LIN {X 0.010,Y -561.070,Z 1059.302,A 0.000,B 0.000,C 90.000,E1 90.286} C_DIS
LIN {X -0.066,Y -561.534,Z 1059.294,A 0.000,B 0.000,C 90.000,E1 88.912} C_DIS
LIN {X -0.024,Y -562.090,Z 1059.285,A 0.000,B 0.000,C 90.000,E1 87.249} C_DIS
LIN {X 0.060,Y -562.761,Z 1059.276,A 0.000,B 0.000,C 90.000,E1 85.584} C_DIS
LIN {X 0.063,Y -563.206,Z 1059.268,A 0.000,B 0.000,C 90.000,E1 84.204} C_DIS
LIN {X -0.191,Y -563.676,Z 1059.257,A 0.000,B 0.000,C 90.000,E1 82.299} C_DIS
LIN {X 0.040,Y -564.205,Z 1059.248,A 0.000,B 0.000,C 90.000,E1 80.622} C_DIS
LIN {X 0.142,Y -565.085,Z 1059.236,A 0.000,B 0.000,C 90.000,E1 78.409} C_DIS
LIN {X -0.127,Y -565.808,Z 1059.228,A 0.000,B 0.000,C 90.000,E1 77.061} C_DIS
LIN {X 0.019,Y -567.276,Z 1059.214,A 0.000,B 0.000,C 90.000,E1 74.574} C_DIS
LIN {X -0.132,Y -568.746,Z 1059.204,A 0.000,B 0.000,C 90.000,E1 72.670} C_DIS
LIN {X -0.096,Y -570.540,Z 1059.192,A 0.000,B 0.000,C 90.000,E1 70.477} C_DIS
LIN {X -0.152,Y -571.474,Z 1059.185,A 0.000,B 0.000,C 90.000,E1 69.390} C_DIS
LIN {X -0.198,Y -572.979,Z 1059.175,A 0.000,B 0.000,C 90.000,E1 67.486} C_DIS
LIN {X -0.127,Y -574.101,Z 1059.166,A 0.000,B 0.000,C 90.000,E1 65.845} C_DIS
LIN {X -0.178,Y -575.248,Z 1059.155,A 0.000,B 0.000,C 90.000,E1 63.948} C_DIS
LIN {X 0.199,Y -576.123,Z 1059.146,A 0.000,B 0.000,C 90.000,E1 62.281} C_DIS
LIN {X 0.224,Y -576.847,Z 1059.139,A 0.000,B 0.000,C 90.000,E1 60.923} C_DIS
LIN {X -0.113,Y -577.556,Z 1059.130,A 0.000,B 0.000,C 90.000,E1 59.331} C_DIS
LIN {X -0.133,Y -578.213,Z 1059.121,A 0.000,B 0.000,C 90.000,E1 57.709} C_DIS
LIN {X -0.146,Y -578.878,Z 1059.112,A 0.000,B 0.000,C 90.000,E1 56.087} C_DIS
LIN {X -0.145,Y -579.399,Z 1059.101,A 0.000,B 0.000,C 90.000,E1 54.196} C_DIS
LIN {X 0.187,Y -579.510,Z 1059.098,A 0.000,B 0.000,C 90.000,E1 53.623} C_DIS
LIN {X 0.206,Y -579.521,Z 1059.091,A 0.000,B 0.000,C 90.000,E1 52.271} C_DIS
LIN {X 0.246,Y -579.470,Z 1059.086,A 0.000,B 0.000,C 90.000,E1 51.457} C_DIS
LIN {X -0.077,Y -579.230,Z 1059.082,A 0.000,B 0.000,C 90.000,E1 50.678} C_DIS
LIN {X 0.207,Y -578.665,Z 1059.074,A 0.000,B 0.000,C 90.000,E1 49.299} C_DIS
LIN {X 0.105,Y -578.034,Z 1059.067,A 0.000,B 0.000,C 90.000,E1 47.957} C_DIS
LIN {X -0.198,Y -577.318,Z 1059.061,A 0.000,B 0.000,C 90.000,E1 46.905} C_DIS
LIN {X 0.198,Y -576.692,Z 1059.056,A 0.000,B 0.000,C 90.000,E1 46.053} C_DIS
LIN {X 0.169,Y -575.894,Z 1059.052,A 0.000,B 0.000,C 90.000,E1 45.243} C_DIS
LIN {X 0.374,Y -574.257,Z 1059.044,A 0.000,B 0.000,C 90.000,E1 43.866} C_DIS
LIN {X 0.147,Y -572.209,Z 1059.036,A 0.000,B 0.000,C 90.000,E1 42.528} C_DIS
LIN {X -0.321,Y -570.874,Z 1059.032,A 0.000,B 0.000,C 90.000,E1 41.757} C_DIS
LIN {X 0.000,Y -569.379,Z 1059.027,A 0.000,B 0.000,C 90.000,E1 40.906} C_DIS
LIN {X -0.265,Y -566.286,Z 1059.020,A 0.000,B 0.000,C 90.000,E1 39.564} C_DIS
LIN {X -0.145,Y -562.491,Z 1059.012,A 0.000,B 0.000,C 90.000,E1 38.177} C_DIS
LIN {X 0.162,Y -559.808,Z 1059.007,A 0.000,B 0.000,C 90.000,E1 37.317} C_DIS
LIN {X -0.096,Y -557.923,Z 1059.004,A 0.000,B 0.000,C 90.000,E1 36.790} C_DIS
LIN {X 0.076,Y -555.871,Z 1059.001,A 0.000,B 0.000,C 90.000,E1 36.217} C_DIS
LIN {X -0.017,Y -552.360,Z 1058.997,A 0.000,B 0.000,C 90.000,E1 35.391} C_DIS
LIN {X -0.014,Y -549.197,Z 1058.993,A 0.000,B 0.000,C 90.000,E1 34.692} C_DIS
LIN {X -0.004,Y -544.551,Z 1058.987,A 0.000,B 0.000,C 90.000,E1 33.706} C_DIS
LIN {X 0.251,Y -538.674,Z 1058.981,A 0.000,B 0.000,C 90.000,E1 32.546} C_DIS
LIN {X -0.167,Y -534.651,Z 1058.977,A 0.000,B 0.000,C 90.000,E1 31.878} C_DIS
LIN {X -0.034,Y -529.513,Z 1058.972,A 0.000,B 0.000,C 90.000,E1 31.003} C_DIS
LIN {X 0.196,Y -524.774,Z 1058.968,A 0.000,B 0.000,C 90.000,E1 30.256} C_DIS
LIN {X -0.212,Y -517.541,Z 1058.963,A 0.000,B 0.000,C 90.000,E1 29.283} C_DIS
LIN {X -0.104,Y -511.824,Z 1058.958,A 0.000,B 0.000,C 90.000,E1 28.537} C_DIS
LIN {X 0.091,Y -506.976,Z 1058.955,A 0.000,B 0.000,C 90.000,E1 27.924} C_DIS
LIN {X -0.206,Y -503.132,Z 1058.953,A 0.000,B 0.000,C 90.000,E1 27.513} C_DIS
LIN {X 0.157,Y -496.395,Z 1058.949,A 0.000,B 0.000,C 90.000,E1 26.744} C_DIS
LIN {X 0.074,Y -490.864,Z 1058.946,A 0.000,B 0.000,C 90.000,E1 26.181} C_DIS
LIN {X 0.160,Y -482.412,Z 1058.941,A 0.000,B 0.000,C 90.000,E1 25.335} C_DIS
LIN {X 0.165,Y -473.830,Z 1058.936,A 0.000,B 0.000,C 90.000,E1 24.515} C_DIS
LIN {X 0.287,Y -466.468,Z 1058.933,A 0.000,B 0.000,C 90.000,E1 23.823} C_DIS
LIN {X 0.179,Y -456.040,Z 1058.928,A 0.000,B 0.000,C 90.000,E1 22.950} C_DIS
LIN {X -0.144,Y -446.987,Z 1058.923,A 0.000,B 0.000,C 90.000,E1 22.206} C_DIS
LIN {X 0.000,Y -427.675,Z 1058.914,A 0.000,B 0.000,C 90.000,E1 20.429} C_DIS
LIN {X -0.121,Y -416.146,Z 1058.907,A 0.000,B 0.000,C 90.000,E1 19.268} C_DIS
LIN {X -0.045,Y -403.587,Z 1058.899,A 0.000,B 0.000,C 90.000,E1 17.819} C_DIS
LIN {X -0.132,Y -398.339,Z 1058.895,A 0.000,B 0.000,C 90.000,E1 17.149} C_DIS
LIN {X -0.196,Y -395.334,Z 1058.893,A 0.000,B 0.000,C 90.000,E1 16.677} C_DIS
LIN {X -0.074,Y -394.456,Z 1058.892,A 0.000,B 0.000,C 90.000,E1 16.496} C_DIS
LIN {X -0.121,Y -392.733,Z 1058.889,A 0.000,B 0.000,C 90.000,E1 16.079} C_DIS
LIN {X 0.029,Y -391.733,Z 1058.886,A 0.000,B 0.000,C 90.000,E1 15.481} C_DIS
LIN {X -0.132,Y -391.606,Z 1058.883,A 0.000,B 0.000,C 90.000,E1 14.883} C_DIS
LIN {X 0.221,Y -392.903,Z 1058.875,A 0.000,B 0.000,C 90.000,E1 13.411} C_DIS
LIN {X -0.007,Y -398.590,Z 1058.853,A 0.000,B 0.000,C 90.000,E1 9.557} C_DIS
LIN {X -0.170,Y -403.813,Z 1058.838,A 0.000,B 0.000,C 90.000,E1 6.777} C_DIS
LIN {X 0.136,Y -409.152,Z 1058.824,A 0.000,B 0.000,C 90.000,E1 4.302} C_DIS
LIN {X 0.131,Y -411.130,Z 1058.820,A 0.000,B 0.000,C 90.000,E1 3.612} C_DIS
LIN {X -0.082,Y -411.998,Z 1058.819,A 0.000,B 0.000,C 90.000,E1 3.383} C_DIS
LIN {X -0.064,Y -415.403,Z 1058.816,A 0.000,B 0.000,C 90.000,E1 2.808} C_DIS
LIN {X -0.061,Y -416.570,Z 1058.815,A 0.000,B 0.000,C 90.000,E1 2.636} C_DIS
LIN {X -0.059,Y -418.064,Z 1058.814,A 0.000,B 0.000,C 90.000,E1 2.465} C_DIS
LIN {X 0.191,Y -421.574,Z 1058.812,A 0.000,B 0.000,C 90.000,E1 2.121} C_DIS
LIN {X 0.026,Y -423.409,Z 1058.811,A 0.000,B 0.000,C 90.000,E1 2.007} C_DIS
LIN {X 0.078,Y -434.006,Z 1058.807,A 0.000,B 0.000,C 90.000,E1 1.318} C_DIS
LIN {X 0.086,Y -456.510,Z 1058.799,A 0.000,B 0.000,C 90.000,E1 359.885} C_DIS
LIN {X 0.073,Y -471.379,Z 1058.794,A 0.000,B 0.000,C 90.000,E1 358.969} C_DIS
LIN {X 0.112,Y -484.516,Z 1058.790,A 0.000,B 0.000,C 90.000,E1 358.165} C_DIS
LIN {X -0.130,Y -495.813,Z 1058.786,A 0.000,B 0.000,C 90.000,E1 357.478} C_DIS
LIN {X -0.216,Y -503.707,Z 1058.783,A 0.000,B 0.000,C 90.000,E1 356.963} C_DIS
LIN {X 0.045,Y -511.351,Z 1058.780,A 0.000,B 0.000,C 90.000,E1 356.388} C_DIS
LIN {X 0.098,Y -518.758,Z 1058.777,A 0.000,B 0.000,C 90.000,E1 355.812} C_DIS
LIN {X -0.107,Y -524.566,Z 1058.774,A 0.000,B 0.000,C 90.000,E1 355.355} C_DIS
LIN {X 0.229,Y -530.049,Z 1058.771,A 0.000,B 0.000,C 90.000,E1 354.837} C_DIS
LIN {X 0.199,Y -535.561,Z 1058.769,A 0.000,B 0.000,C 90.000,E1 354.318} C_DIS
LIN {X -0.151,Y -541.884,Z 1058.765,A 0.000,B 0.000,C 90.000,E1 353.685} C_DIS
LIN {X 0.069,Y -546.768,Z 1058.762,A 0.000,B 0.000,C 90.000,E1 353.109} C_DIS
LIN {X 0.008,Y -552.220,Z 1058.758,A 0.000,B 0.000,C 90.000,E1 352.413} C_DIS
LIN {X 0.161,Y -556.239,Z 1058.755,A 0.000,B 0.000,C 90.000,E1 351.837} C_DIS
LIN {X 0.178,Y -560.694,Z 1058.751,A 0.000,B 0.000,C 90.000,E1 351.141} C_DIS
LIN {X -0.168,Y -564.024,Z 1058.748,A 0.000,B 0.000,C 90.000,E1 350.622} C_DIS
LIN {X -0.088,Y -567.760,Z 1058.744,A 0.000,B 0.000,C 90.000,E1 349.926} C_DIS
LIN {X 0.134,Y -571.203,Z 1058.740,A 0.000,B 0.000,C 90.000,E1 349.218} C_DIS
LIN {X 0.044,Y -575.033,Z 1058.736,A 0.000,B 0.000,C 90.000,E1 348.409} C_DIS
LIN {X 0.204,Y -580.307,Z 1058.729,A 0.000,B 0.000,C 90.000,E1 347.173} C_DIS
LIN {X -0.019,Y -584.594,Z 1058.723,A 0.000,B 0.000,C 90.000,E1 346.117} C_DIS
LIN {X 0.204,Y -589.665,Z 1058.715,A 0.000,B 0.000,C 90.000,E1 344.755} C_DIS
LIN {X -0.056,Y -594.516,Z 1058.708,A 0.000,B 0.000,C 90.000,E1 343.449} C_DIS
LIN {X 0.229,Y -598.177,Z 1058.702,A 0.000,B 0.000,C 90.000,E1 342.362} C_DIS
LIN {X 0.003,Y -601.590,Z 1058.696,A 0.000,B 0.000,C 90.000,E1 341.329} C_DIS
LIN {X -0.091,Y -603.905,Z 1058.692,A 0.000,B 0.000,C 90.000,E1 340.550} C_DIS
LIN {X 0.038,Y -606.170,Z 1058.688,A 0.000,B 0.000,C 90.000,E1 339.752} C_DIS
LIN {X -0.141,Y -609.589,Z 1058.680,A 0.000,B 0.000,C 90.000,E1 338.465} C_DIS
LIN {X 0.049,Y -611.504,Z 1058.676,A 0.000,B 0.000,C 90.000,E1 337.667} C_DIS
LIN {X 0.187,Y -614.433,Z 1058.669,A 0.000,B 0.000,C 90.000,E1 336.357} C_DIS
LIN {X -0.191,Y -616.880,Z 1058.662,A 0.000,B 0.000,C 90.000,E1 335.101} C_DIS
LIN {X 0.291,Y -618.961,Z 1058.654,A 0.000,B 0.000,C 90.000,E1 333.768} C_DIS
LIN {X 0.251,Y -620.720,Z 1058.647,A 0.000,B 0.000,C 90.000,E1 332.487} C_DIS
LIN {X -0.316,Y -622.272,Z 1058.640,A 0.000,B 0.000,C 90.000,E1 331.257} C_DIS
LIN {X -0.017,Y -623.078,Z 1058.636,A 0.000,B 0.000,C 90.000,E1 330.461} C_DIS
LIN {X -0.243,Y -623.905,Z 1058.630,A 0.000,B 0.000,C 90.000,E1 329.459} C_DIS
LIN {X 0.075,Y -624.459,Z 1058.625,A 0.000,B 0.000,C 90.000,E1 328.408} C_DIS
LIN {X -0.134,Y -624.866,Z 1058.620,A 0.000,B 0.000,C 90.000,E1 327.661} C_DIS
LIN {X -0.006,Y -624.992,Z 1058.615,A 0.000,B 0.000,C 90.000,E1 326.628} C_DIS
LIN {X 0.126,Y -624.944,Z 1058.609,A 0.000,B 0.000,C 90.000,E1 325.595} C_DIS
LIN {X 0.084,Y -624.711,Z 1058.602,A 0.000,B 0.000,C 90.000,E1 324.322} C_DIS
LIN {X 0.178,Y -624.070,Z 1058.591,A 0.000,B 0.000,C 90.000,E1 322.271} C_DIS
LIN {X -0.171,Y -623.409,Z 1058.576,A 0.000,B 0.000,C 90.000,E1 319.747} C_DIS
LIN {X 0.056,Y -623.246,Z 1058.569,A 0.000,B 0.000,C 90.000,E1 318.447} C_DIS
LIN {X 0.098,Y -623.046,Z 1058.565,A 0.000,B 0.000,C 90.000,E1 317.676} C_DIS
LIN {X -0.110,Y -622.573,Z 1058.554,A 0.000,B 0.000,C 90.000,E1 315.648} C_DIS
LIN {X -0.212,Y -622.237,Z 1058.544,A 0.000,B 0.000,C 90.000,E1 313.866} C_DIS
LIN {X -0.185,Y -622.125,Z 1058.539,A 0.000,B 0.000,C 90.000,E1 313.095} C_DIS
LIN {X 0.433,Y -621.704,Z 1058.532,A 0.000,B 0.000,C 90.000,E1 311.757} C_DIS
LIN {X -0.254,Y -621.130,Z 1058.525,A 0.000,B 0.000,C 90.000,E1 310.539} C_DIS
LIN {X 0.066,Y -621.133,Z 1058.524,A 0.000,B 0.000,C 90.000,E1 310.253} C_DIS
LIN {X 0.235,Y -620.888,Z 1058.521,A 0.000,B 0.000,C 90.000,E1 309.725} C_DIS
LIN {X 0.078,Y -620.896,Z 1058.519,A 0.000,B 0.000,C 90.000,E1 309.483} C_DIS
LIN {X -0.284,Y -620.114,Z 1058.505,A 0.000,B 0.000,C 90.000,E1 306.950} C_DIS
LIN {X -0.138,Y -620.085,Z 1058.502,A 0.000,B 0.000,C 90.000,E1 306.423} C_DIS
LIN {X -0.083,Y -619.896,Z 1058.497,A 0.000,B 0.000,C 90.000,E1 305.391} C_DIS
LIN {X 0.238,Y -619.761,Z 1058.495,A 0.000,B 0.000,C 90.000,E1 305.105} C_DIS
LIN {X 0.013,Y -619.990,Z 1058.492,A 0.000,B 0.000,C 90.000,E1 304.612} C_DIS
LIN {X 0.393,Y -619.920,Z 1058.485,A 0.000,B 0.000,C 90.000,E1 303.293} C_DIS
LIN {X -0.151,Y -619.823,Z 1058.484,A 0.000,B 0.000,C 90.000,E1 303.086} C_DIS
LIN {X 0.139,Y -620.073,Z 1058.481,A 0.000,B 0.000,C 90.000,E1 302.546} C_DIS
LIN {X -0.113,Y -620.174,Z 1058.477,A 0.000,B 0.000,C 90.000,E1 301.799} C_DIS
LIN {X 0.165,Y -620.036,Z 1058.472,A 0.000,B 0.000,C 90.000,E1 301.003} C_DIS
LIN {X -0.090,Y -620.335,Z 1058.468,A 0.000,B 0.000,C 90.000,E1 300.256} C_DIS
LIN {X 0.167,Y -620.678,Z 1058.460,A 0.000,B 0.000,C 90.000,E1 298.693} C_DIS
LIN {X -0.120,Y -620.453,Z 1058.451,A 0.000,B 0.000,C 90.000,E1 297.180} C_DIS
LIN {X -0.149,Y -619.802,Z 1058.444,A 0.000,B 0.000,C 90.000,E1 295.899} C_DIS
LIN {X 0.115,Y -618.831,Z 1058.438,A 0.000,B 0.000,C 90.000,E1 294.847} C_DIS
LIN {X 0.082,Y -617.754,Z 1058.434,A 0.000,B 0.000,C 90.000,E1 294.079} C_DIS
LIN {X -0.236,Y -615.850,Z 1058.428,A 0.000,B 0.000,C 90.000,E1 293.078} C_DIS
LIN {X 0.281,Y -614.623,Z 1058.425,A 0.000,B 0.000,C 90.000,E1 292.514} C_DIS
LIN {X -0.014,Y -612.935,Z 1058.422,A 0.000,B 0.000,C 90.000,E1 292.025} C_DIS
LIN {X -0.050,Y -611.999,Z 1058.421,A 0.000,B 0.000,C 90.000,E1 291.770} C_DIS
LIN {X 0.210,Y -609.689,Z 1058.418,A 0.000,B 0.000,C 90.000,E1 291.227} C_DIS
LIN {X -0.112,Y -606.397,Z 1058.415,A 0.000,B 0.000,C 90.000,E1 290.737} C_DIS
LIN {X -0.287,Y -601.104,Z 1058.412,A 0.000,B 0.000,C 90.000,E1 290.248} C_DIS
LIN {X -0.092,Y -596.948,Z 1058.410,A 0.000,B 0.000,C 90.000,E1 289.866} C_DIS
LIN {X -0.208,Y -595.289,Z 1058.410,A 0.000,B 0.000,C 90.000,E1 289.758} C_DIS
LIN {X 0.152,Y -588.650,Z 1058.407,A 0.000,B 0.000,C 90.000,E1 289.322} C_DIS
LIN {X 0.358,Y -581.461,Z 1058.406,A 0.000,B 0.000,C 90.000,E1 288.960} C_DIS
LIN {X 0.216,Y -570.740,Z 1058.403,A 0.000,B 0.000,C 90.000,E1 288.544} C_DIS
LIN {X -0.092,Y -560.846,Z 1058.402,A 0.000,B 0.000,C 90.000,E1 288.362} C_DIS
LIN {X -0.097,Y -556.775,Z 1058.402,A 0.000,B 0.000,C 90.000,E1 288.290} C_DIS
LIN {X 0.284,Y -550.568,Z 1058.401,A 0.000,B 0.000,C 90.000,E1 288.236} C_DIS
LIN {X -0.233,Y -547.940,Z 1058.401,A 0.000,B 0.000,C 90.000,E1 288.236} C_DIS
LIN {X 0.243,Y -547.765,Z 1058.401,A 0.000,B 0.000,C 90.000,E1 288.181} C_DIS
LIN {X -0.099,Y -546.592,Z 1058.400,A 0.000,B 0.000,C 90.000,E1 287.946} C_DIS
LIN {X 0.275,Y -546.226,Z 1058.399,A 0.000,B 0.000,C 90.000,E1 287.819} C_DIS
LIN {X -0.166,Y -545.992,Z 1058.398,A 0.000,B 0.000,C 90.000,E1 287.583} C_DIS
LIN {X 0.079,Y -545.427,Z 1058.396,A 0.000,B 0.000,C 90.000,E1 287.275} C_DIS
LIN {X 0.231,Y -544.728,Z 1058.382,A 0.000,B 0.000,C 90.000,E1 284.717} C_DIS
LIN {X -0.256,Y -544.250,Z 1058.374,A 0.000,B 0.000,C 90.000,E1 283.355} C_DIS
LIN {X 0.186,Y -543.503,Z 1058.366,A 0.000,B 0.000,C 90.000,E1 281.895} C_DIS
LIN {X 0.170,Y -542.509,Z 1058.357,A 0.000,B 0.000,C 90.000,E1 280.197} C_DIS
LIN {X 0.027,Y -541.501,Z 1058.347,A 0.000,B 0.000,C 90.000,E1 278.511} C_DIS
LIN {X -0.221,Y -540.467,Z 1058.338,A 0.000,B 0.000,C 90.000,E1 276.834} C_DIS
LIN {X -0.084,Y -539.816,Z 1058.332,A 0.000,B 0.000,C 90.000,E1 275.682} C_DIS
LIN {X 0.109,Y -538.669,Z 1058.321,A 0.000,B 0.000,C 90.000,E1 273.669} C_DIS
LIN {X 0.230,Y -537.557,Z 1058.309,A 0.000,B 0.000,C 90.000,E1 271.661} C_DIS
LIN {X 0.266,Y -536.897,Z 1058.303,A 0.000,B 0.000,C 90.000,E1 270.516} C_DIS
LIN {X -0.228,Y -535.841,Z 1058.294,A 0.000,B 0.000,C 90.000,E1 268.854} C_DIS
LIN {X -0.200,Y -535.169,Z 1058.287,A 0.000,B 0.000,C 90.000,E1 267.707} C_DIS
LIN {X -0.183,Y -534.244,Z 1058.279,A 0.000,B 0.000,C 90.000,E1 266.274} C_DIS
LIN {X -0.152,Y -533.229,Z 1058.271,A 0.000,B 0.000,C 90.000,E1 264.837} C_DIS
LIN {X -0.084,Y -532.096,Z 1058.263,A 0.000,B 0.000,C 90.000,E1 263.394} C_DIS
LIN {X -0.038,Y -531.301,Z 1058.259,A 0.000,B 0.000,C 90.000,E1 262.527} C_DIS
LIN {X 0.031,Y -528.529,Z 1058.244,A 0.000,B 0.000,C 90.000,E1 259.926} C_DIS
LIN {X 0.172,Y -526.943,Z 1058.236,A 0.000,B 0.000,C 90.000,E1 258.465} C_DIS
LIN {X -0.232,Y -525.359,Z 1058.228,A 0.000,B 0.000,C 90.000,E1 257.061} C_DIS
LIN {X 0.112,Y -523.228,Z 1058.217,A 0.000,B 0.000,C 90.000,E1 254.991} C_DIS
LIN {X -0.099,Y -521.731,Z 1058.209,A 0.000,B 0.000,C 90.000,E1 253.559} C_DIS
LIN {X 0.173,Y -520.525,Z 1058.202,A 0.000,B 0.000,C 90.000,E1 252.362} C_DIS
LIN {X 0.210,Y -518.553,Z 1058.192,A 0.000,B 0.000,C 90.000,E1 250.604} C_DIS
LIN {X -0.151,Y -516.089,Z 1058.181,A 0.000,B 0.000,C 90.000,E1 248.592} C_DIS
LIN {X 0.027,Y -514.095,Z 1058.173,A 0.000,B 0.000,C 90.000,E1 247.102} C_DIS
LIN {X -0.073,Y -512.845,Z 1058.168,A 0.000,B 0.000,C 90.000,E1 246.230} C_DIS
LIN {X 0.250,Y -510.654,Z 1058.160,A 0.000,B 0.000,C 90.000,E1 244.717} C_DIS
LIN {X 0.066,Y -508.210,Z 1058.151,A 0.000,B 0.000,C 90.000,E1 243.256} C_DIS
LIN {X -0.253,Y -506.287,Z 1058.145,A 0.000,B 0.000,C 90.000,E1 242.103} C_DIS
LIN {X -0.051,Y -503.777,Z 1058.137,A 0.000,B 0.000,C 90.000,E1 240.589} C_DIS
LIN {X 0.103,Y -500.991,Z 1058.128,A 0.000,B 0.000,C 90.000,E1 239.076} C_DIS
LIN {X 0.033,Y -498.256,Z 1058.120,A 0.000,B 0.000,C 90.000,E1 237.582} C_DIS
LIN {X 0.052,Y -495.975,Z 1058.113,A 0.000,B 0.000,C 90.000,E1 236.373} C_DIS
LIN {X -0.139,Y -491.780,Z 1058.101,A 0.000,B 0.000,C 90.000,E1 234.276} C_DIS
LIN {X 0.092,Y -489.741,Z 1058.096,A 0.000,B 0.000,C 90.000,E1 233.336} C_DIS
LIN {X 0.316,Y -484.801,Z 1058.085,A 0.000,B 0.000,C 90.000,E1 231.170} C_DIS
LIN {X -0.158,Y -480.608,Z 1058.074,A 0.000,B 0.000,C 90.000,E1 229.380} C_DIS
LIN {X 0.266,Y -476.716,Z 1058.064,A 0.000,B 0.000,C 90.000,E1 227.472} C_DIS
LIN {X -0.201,Y -473.590,Z 1058.055,A 0.000,B 0.000,C 90.000,E1 225.972} C_DIS
LIN {X 0.185,Y -471.218,Z 1058.048,A 0.000,B 0.000,C 90.000,E1 224.676} C_DIS
LIN {X -0.226,Y -466.856,Z 1058.036,A 0.000,B 0.000,C 90.000,E1 222.528} C_DIS
LIN {X -0.122,Y -463.054,Z 1058.026,A 0.000,B 0.000,C 90.000,E1 220.620} C_DIS
LIN {X -0.050,Y -459.058,Z 1058.015,A 0.000,B 0.000,C 90.000,E1 218.705} C_DIS
LIN {X 0.020,Y -454.530,Z 1058.003,A 0.000,B 0.000,C 90.000,E1 216.457} C_DIS
LIN {X 0.259,Y -451.211,Z 1057.994,A 0.000,B 0.000,C 90.000,E1 214.818} C_DIS
LIN {X -0.068,Y -446.460,Z 1057.981,A 0.000,B 0.000,C 90.000,E1 212.594} C_DIS
LIN {X 0.192,Y -443.759,Z 1057.974,A 0.000,B 0.000,C 90.000,E1 211.258} C_DIS
LIN {X -0.099,Y -439.661,Z 1057.963,A 0.000,B 0.000,C 90.000,E1 209.333} C_DIS
LIN {X 0.112,Y -434.186,Z 1057.948,A 0.000,B 0.000,C 90.000,E1 206.668} C_DIS
LIN {X -0.037,Y -430.849,Z 1057.939,A 0.000,B 0.000,C 90.000,E1 205.027} C_DIS
LIN {X 0.103,Y -424.745,Z 1057.921,A 0.000,B 0.000,C 90.000,E1 201.663} C_DIS
LIN {X -0.043,Y -421.218,Z 1057.907,A 0.000,B 0.000,C 90.000,E1 199.322} C_DIS
LIN {X -0.107,Y -419.525,Z 1057.898,A 0.000,B 0.000,C 90.000,E1 197.638} C_DIS
LIN {X -0.129,Y -418.915,Z 1057.892,A 0.000,B 0.000,C 90.000,E1 196.622} C_DIS
LIN {X -0.156,Y -418.763,Z 1057.887,A 0.000,B 0.000,C 90.000,E1 195.607} C_DIS
LIN {X 0.218,Y -419.505,Z 1057.881,A 0.000,B 0.000,C 90.000,E1 194.537} C_DIS
LIN {X -0.133,Y -419.914,Z 1057.879,A 0.000,B 0.000,C 90.000,E1 194.245} C_DIS
LIN {X 0.089,Y -421.185,Z 1057.875,A 0.000,B 0.000,C 90.000,E1 193.536} C_DIS
LIN {X -0.009,Y -423.685,Z 1057.871,A 0.000,B 0.000,C 90.000,E1 192.703} C_DIS
LIN {X -0.176,Y -428.006,Z 1057.865,A 0.000,B 0.000,C 90.000,E1 191.715} C_DIS
LIN {X -0.185,Y -434.354,Z 1057.859,A 0.000,B 0.000,C 90.000,E1 190.546} C_DIS
LIN {X 0.093,Y -444.479,Z 1057.849,A 0.000,B 0.000,C 90.000,E1 188.859} C_DIS
LIN {X -0.003,Y -454.003,Z 1057.841,A 0.000,B 0.000,C 90.000,E1 187.409} C_DIS
LIN {X 0.135,Y -460.315,Z 1057.836,A 0.000,B 0.000,C 90.000,E1 186.429} C_DIS
LIN {X 0.199,Y -465.502,Z 1057.831,A 0.000,B 0.000,C 90.000,E1 185.625} C_DIS
LIN {X -0.146,Y -470.486,Z 1057.827,A 0.000,B 0.000,C 90.000,E1 184.878} C_DIS
LIN {X -0.162,Y -477.151,Z 1057.821,A 0.000,B 0.000,C 90.000,E1 183.784} C_DIS
LIN {X -0.122,Y -483.716,Z 1057.815,A 0.000,B 0.000,C 90.000,E1 182.694} C_DIS
LIN {X 0.003,Y -490.101,Z 1057.809,A 0.000,B 0.000,C 90.000,E1 181.604} C_DIS
LIN {X -0.068,Y -499.824,Z 1057.800,A 0.000,B 0.000,C 90.000,E1 179.943} C_DIS
LIN {X 0.158,Y -507.412,Z 1057.792,A 0.000,B 0.000,C 90.000,E1 178.568} C_DIS
LIN {X -0.197,Y -514.046,Z 1057.786,A 0.000,B 0.000,C 90.000,E1 177.421} C_DIS
LIN {X 0.034,Y -522.154,Z 1057.777,A 0.000,B 0.000,C 90.000,E1 175.927} C_DIS
LIN {X 0.130,Y -529.318,Z 1057.770,A 0.000,B 0.000,C 90.000,E1 174.609} C_DIS
LIN {X 0.126,Y -535.565,Z 1057.764,A 0.000,B 0.000,C 90.000,E1 173.457} C_DIS
LIN {X 0.082,Y -544.009,Z 1057.755,A 0.000,B 0.000,C 90.000,E1 171.894} C_DIS
LIN {X -0.070,Y -551.561,Z 1057.747,A 0.000,B 0.000,C 90.000,E1 170.500} C_DIS
LIN {X 0.033,Y -556.693,Z 1057.742,A 0.000,B 0.000,C 90.000,E1 169.511} C_DIS
LIN {X -0.205,Y -561.051,Z 1057.737,A 0.000,B 0.000,C 90.000,E1 168.701} C_DIS
LIN {X -0.261,Y -567.274,Z 1057.730,A 0.000,B 0.000,C 90.000,E1 167.465} C_DIS
LIN {X -0.096,Y -572.716,Z 1057.724,A 0.000,B 0.000,C 90.000,E1 166.353} C_DIS
LIN {X 0.077,Y -576.568,Z 1057.720,A 0.000,B 0.000,C 90.000,E1 165.519} C_DIS
LIN {X -0.290,Y -582.172,Z 1057.713,A 0.000,B 0.000,C 90.000,E1 164.338} C_DIS
LIN {X 0.133,Y -587.439,Z 1057.706,A 0.000,B 0.000,C 90.000,E1 163.087} C_DIS
LIN {X -0.241,Y -591.929,Z 1057.700,A 0.000,B 0.000,C 90.000,E1 162.054} C_DIS
LIN {X 0.016,Y -596.026,Z 1057.694,A 0.000,B 0.000,C 90.000,E1 160.967} C_DIS
LIN {X -0.234,Y -599.934,Z 1057.688,A 0.000,B 0.000,C 90.000,E1 159.934} C_DIS
LIN {X 0.124,Y -603.658,Z 1057.683,A 0.000,B 0.000,C 90.000,E1 158.847} C_DIS
LIN {X 0.126,Y -607.967,Z 1057.675,A 0.000,B 0.000,C 90.000,E1 157.539} C_DIS
LIN {X 0.209,Y -611.893,Z 1057.668,A 0.000,B 0.000,C 90.000,E1 156.230} C_DIS
LIN {X -0.179,Y -614.885,Z 1057.662,A 0.000,B 0.000,C 90.000,E1 155.229} C_DIS
LIN {X 0.273,Y -618.408,Z 1057.655,A 0.000,B 0.000,C 90.000,E1 153.896} C_DIS
LIN {X 0.229,Y -621.721,Z 1057.648,A 0.000,B 0.000,C 90.000,E1 152.615} C_DIS
LIN {X -0.009,Y -625.464,Z 1057.640,A 0.000,B 0.000,C 90.000,E1 151.101} C_DIS
LIN {X 0.045,Y -628.493,Z 1057.632,A 0.000,B 0.000,C 90.000,E1 149.822} C_DIS
LIN {X -0.131,Y -630.323,Z 1057.628,A 0.000,B 0.000,C 90.000,E1 149.076} C_DIS
LIN {X 0.114,Y -633.680,Z 1057.620,A 0.000,B 0.000,C 90.000,E1 147.533} C_DIS
LIN {X 0.241,Y -636.974,Z 1057.611,A 0.000,B 0.000,C 90.000,E1 146.008} C_DIS
LIN {X 0.044,Y -639.668,Z 1057.604,A 0.000,B 0.000,C 90.000,E1 144.769} C_DIS
LIN {X -0.150,Y -641.796,Z 1057.599,A 0.000,B 0.000,C 90.000,E1 143.783} C_DIS
LIN {X -0.097,Y -645.552,Z 1057.589,A 0.000,B 0.000,C 90.000,E1 142.029} C_DIS
LIN {X -0.304,Y -648.180,Z 1057.582,A 0.000,B 0.000,C 90.000,E1 140.803} C_DIS
LIN {X -0.125,Y -651.385,Z 1057.574,A 0.000,B 0.000,C 90.000,E1 139.299} C_DIS
LIN {X 0.070,Y -655.128,Z 1057.564,A 0.000,B 0.000,C 90.000,E1 137.553} C_DIS
LIN {X 0.311,Y -659.077,Z 1057.555,A 0.000,B 0.000,C 90.000,E1 135.810} C_DIS
LIN {X 0.137,Y -665.992,Z 1057.540,A 0.000,B 0.000,C 90.000,E1 133.137} C_DIS
LIN {X 0.168,Y -669.259,Z 1057.533,A 0.000,B 0.000,C 90.000,E1 131.919} C_DIS
LIN {X -0.155,Y -673.765,Z 1057.524,A 0.000,B 0.000,C 90.000,E1 130.253} C_DIS
LIN {X -0.406,Y -677.608,Z 1057.516,A 0.000,B 0.000,C 90.000,E1 128.830} C_DIS
LIN {X -0.085,Y -680.720,Z 1057.509,A 0.000,B 0.000,C 90.000,E1 127.604} C_DIS
LIN {X -0.069,Y -684.966,Z 1057.500,A 0.000,B 0.000,C 90.000,E1 125.931} C_DIS
LIN {X -0.036,Y -687.949,Z 1057.493,A 0.000,B 0.000,C 90.000,E1 124.739} C_DIS
LIN {X -0.107,Y -692.034,Z 1057.484,A 0.000,B 0.000,C 90.000,E1 123.086} C_DIS
LIN {X 0.240,Y -694.825,Z 1057.477,A 0.000,B 0.000,C 90.000,E1 121.878} C_DIS
LIN {X 0.041,Y -697.509,Z 1057.471,A 0.000,B 0.000,C 90.000,E1 120.718} C_DIS
LIN {X -0.141,Y -699.335,Z 1057.465,A 0.000,B 0.000,C 90.000,E1 119.795} C_DIS
LIN {X 0.044,Y -700.455,Z 1057.462,A 0.000,B 0.000,C 90.000,E1 119.077} C_DIS
LIN {X -0.030,Y -701.009,Z 1057.459,A 0.000,B 0.000,C 90.000,E1 118.615} C_DIS
LIN {X 0.271,Y -703.133,Z 1057.447,A 0.000,B 0.000,C 90.000,E1 116.488} C_DIS
LIN {X -0.172,Y -704.013,Z 1057.442,A 0.000,B 0.000,C 90.000,E1 115.591} C_DIS
LIN {X -0.255,Y -704.460,Z 1057.438,A 0.000,B 0.000,C 90.000,E1 114.899} C_DIS
LIN {X 0.030,Y -704.553,Z 1057.437,A 0.000,B 0.000,C 90.000,E1 114.643} C_DIS
LIN {X -0.332,Y -704.310,Z 1057.434,A 0.000,B 0.000,C 90.000,E1 114.207} C_DIS
LIN {X -0.048,Y -703.973,Z 1057.433,A 0.000,B 0.000,C 90.000,E1 113.951} C_DIS
LIN {X 0.233,Y -702.696,Z 1057.431,A 0.000,B 0.000,C 90.000,E1 113.462} C_DIS
LIN {X -0.134,Y -701.552,Z 1057.429,A 0.000,B 0.000,C 90.000,E1 113.259} C_DIS
LIN {X 0.134,Y -698.263,Z 1057.427,A 0.000,B 0.000,C 90.000,E1 112.770} C_DIS
LIN {X 0.264,Y -697.093,Z 1057.426,A 0.000,B 0.000,C 90.000,E1 112.642} C_DIS
LIN {X 0.393,Y -695.284,Z 1057.425,A 0.000,B 0.000,C 90.000,E1 112.514} C_DIS
LIN {X 0.047,Y -688.046,Z 1057.423,A 0.000,B 0.000,C 90.000,E1 112.206} C_DIS
LIN {X 0.236,Y -684.686,Z 1057.423,A 0.000,B 0.000,C 90.000,E1 112.078} C_DIS
LIN {X 0.133,Y -675.816,Z 1057.422,A 0.000,B 0.000,C 90.000,E1 111.972} C_DIS
LIN {X 0.072,Y -609.219,Z 1057.422,A 0.000,B 0.000,C 90.000,E1 111.972} C_DIS
LIN {X -0.050,Y -605.267,Z 1057.421,A 0.000,B 0.000,C 90.000,E1 111.844} C_DIS
LIN {X 0.304,Y -603.017,Z 1057.421,A 0.000,B 0.000,C 90.000,E1 111.716} C_DIS
LIN {X 0.256,Y -597.192,Z 1057.419,A 0.000,B 0.000,C 90.000,E1 111.408} C_DIS
LIN {X 0.040,Y -591.756,Z 1057.417,A 0.000,B 0.000,C 90.000,E1 111.046} C_DIS
LIN {X 0.215,Y -578.536,Z 1057.411,A 0.000,B 0.000,C 90.000,E1 109.939} C_DIS
LIN {X -0.179,Y -574.166,Z 1057.409,A 0.000,B 0.000,C 90.000,E1 109.631} C_DIS
LIN {X 0.082,Y -569.684,Z 1057.407,A 0.000,B 0.000,C 90.000,E1 109.268} C_DIS
LIN {X 0.015,Y -564.472,Z 1057.405,A 0.000,B 0.000,C 90.000,E1 108.960} C_DIS
LIN {X 0.107,Y -553.356,Z 1057.402,A 0.000,B 0.000,C 90.000,E1 108.308} C_DIS
LIN {X 0.164,Y -549.583,Z 1057.400,A 0.000,B 0.000,C 90.000,E1 108.055} C_DIS
LIN {X -0.083,Y -547.858,Z 1057.399,A 0.000,B 0.000,C 90.000,E1 107.873} C_DIS
LIN {X 0.271,Y -547.723,Z 1057.399,A 0.000,B 0.000,C 90.000,E1 107.819} C_DIS
LIN {X 0.229,Y -547.695,Z 1057.399,A 0.000,B 0.000,C 90.000,E1 107.819} C_DIS
LIN {X -0.331,Y -547.249,Z 1057.398,A 0.000,B 0.000,C 90.000,E1 107.583} C_DIS
LIN {X 0.204,Y -548.641,Z 1057.384,A 0.000,B 0.000,C 90.000,E1 105.134} C_DIS
LIN {X 0.240,Y -550.164,Z 1057.372,A 0.000,B 0.000,C 90.000,E1 102.883} C_DIS
LIN {X -0.050,Y -551.883,Z 1057.361,A 0.000,B 0.000,C 90.000,E1 100.950} C_DIS
LIN {X 0.177,Y -554.268,Z 1057.348,A 0.000,B 0.000,C 90.000,E1 98.690} C_DIS
LIN {X 0.047,Y -555.510,Z 1057.342,A 0.000,B 0.000,C 90.000,E1 97.587} C_DIS
LIN {X -0.015,Y -557.171,Z 1057.334,A 0.000,B 0.000,C 90.000,E1 96.201} C_DIS
LIN {X -0.180,Y -558.299,Z 1057.328,A 0.000,B 0.000,C 90.000,E1 95.106} C_DIS
LIN {X 0.099,Y -558.963,Z 1057.324,A 0.000,B 0.000,C 90.000,E1 94.245} C_DIS
LIN {X -0.083,Y -559.752,Z 1057.318,A 0.000,B 0.000,C 90.000,E1 93.154} C_DIS
LIN {X -0.144,Y -560.438,Z 1057.310,A 0.000,B 0.000,C 90.000,E1 91.776} C_DIS
LIN {X -0.138,Y -561.118,Z 1057.301,A 0.000,B 0.000,C 90.000,E1 90.115} C_DIS
LIN {X -0.214,Y -561.549,Z 1057.293,A 0.000,B 0.000,C 90.000,E1 88.740} C_DIS
LIN {X -0.174,Y -562.091,Z 1057.284,A 0.000,B 0.000,C 90.000,E1 87.078} C_DIS
LIN {X -0.186,Y -562.703,Z 1057.276,A 0.000,B 0.000,C 90.000,E1 85.698} C_DIS
LIN {X -0.184,Y -563.124,Z 1057.268,A 0.000,B 0.000,C 90.000,E1 84.318} C_DIS
LIN {X 0.124,Y -563.592,Z 1057.258,A 0.000,B 0.000,C 90.000,E1 82.356} C_DIS
LIN {X -0.200,Y -564.122,Z 1057.248,A 0.000,B 0.000,C 90.000,E1 80.735} C_DIS
LIN {X 0.074,Y -565.114,Z 1057.235,A 0.000,B 0.000,C 90.000,E1 78.229} C_DIS
LIN {X -0.190,Y -565.831,Z 1057.227,A 0.000,B 0.000,C 90.000,E1 76.881} C_DIS
LIN {X -0.206,Y -567.154,Z 1057.215,A 0.000,B 0.000,C 90.000,E1 74.685} C_DIS
LIN {X 0.194,Y -568.616,Z 1057.204,A 0.000,B 0.000,C 90.000,E1 72.725} C_DIS
LIN {X 0.042,Y -570.402,Z 1057.192,A 0.000,B 0.000,C 90.000,E1 70.550} C_DIS
LIN {X -0.203,Y -571.541,Z 1057.184,A 0.000,B 0.000,C 90.000,E1 69.209} C_DIS
LIN {X 0.138,Y -572.834,Z 1057.175,A 0.000,B 0.000,C 90.000,E1 67.539} C_DIS
LIN {X -0.183,Y -574.144,Z 1057.165,A 0.000,B 0.000,C 90.000,E1 65.665} C_DIS
LIN {X -0.240,Y -575.229,Z 1057.154,A 0.000,B 0.000,C 90.000,E1 63.768} C_DIS
LIN {X -0.078,Y -575.813,Z 1057.148,A 0.000,B 0.000,C 90.000,E1 62.666} C_DIS
LIN {X -0.208,Y -576.673,Z 1057.139,A 0.000,B 0.000,C 90.000,E1 61.051} C_DIS
LIN {X -0.049,Y -577.376,Z 1057.130,A 0.000,B 0.000,C 90.000,E1 59.410} C_DIS
LIN {X -0.071,Y -577.803,Z 1057.124,A 0.000,B 0.000,C 90.000,E1 58.329} C_DIS
LIN {X -0.085,Y -578.254,Z 1057.118,A 0.000,B 0.000,C 90.000,E1 57.248} C_DIS
LIN {X 0.060,Y -578.748,Z 1057.110,A 0.000,B 0.000,C 90.000,E1 55.881} C_DIS
LIN {X 0.056,Y -579.295,Z 1057.100,A 0.000,B 0.000,C 90.000,E1 53.989} C_DIS
LIN {X -0.095,Y -579.337,Z 1057.094,A 0.000,B 0.000,C 90.000,E1 52.924} C_DIS
LIN {X 0.271,Y -579.266,Z 1057.087,A 0.000,B 0.000,C 90.000,E1 51.537} C_DIS
LIN {X 0.310,Y -579.046,Z 1057.082,A 0.000,B 0.000,C 90.000,E1 50.723} C_DIS
LIN {X 0.223,Y -578.450,Z 1057.074,A 0.000,B 0.000,C 90.000,E1 49.380} C_DIS
LIN {X -0.313,Y -577.813,Z 1057.067,A 0.000,B 0.000,C 90.000,E1 48.081} C_DIS
LIN {X -0.191,Y -577.109,Z 1057.061,A 0.000,B 0.000,C 90.000,E1 46.986} C_DIS
LIN {X -0.079,Y -576.201,Z 1057.055,A 0.000,B 0.000,C 90.000,E1 45.891} C_DIS
LIN {X -0.112,Y -575.348,Z 1057.050,A 0.000,B 0.000,C 90.000,E1 45.081} C_DIS
LIN {X 0.372,Y -574.002,Z 1057.044,A 0.000,B 0.000,C 90.000,E1 43.947} C_DIS
LIN {X 0.017,Y -572.354,Z 1057.038,A 0.000,B 0.000,C 90.000,E1 42.894} C_DIS
LIN {X -0.030,Y -571.057,Z 1057.034,A 0.000,B 0.000,C 90.000,E1 42.081} C_DIS
LIN {X -0.010,Y -569.094,Z 1057.028,A 0.000,B 0.000,C 90.000,E1 40.987} C_DIS
LIN {X -0.079,Y -567.252,Z 1057.023,A 0.000,B 0.000,C 90.000,E1 40.172} C_DIS
LIN {X -0.163,Y -565.260,Z 1057.019,A 0.000,B 0.000,C 90.000,E1 39.358} C_DIS
LIN {X -0.161,Y -562.183,Z 1057.012,A 0.000,B 0.000,C 90.000,E1 38.257} C_DIS
LIN {X -0.301,Y -559.493,Z 1057.008,A 0.000,B 0.000,C 90.000,E1 37.443} C_DIS
LIN {X -0.115,Y -557.565,Z 1057.005,A 0.000,B 0.000,C 90.000,E1 36.870} C_DIS
LIN {X 0.135,Y -554.412,Z 1057.000,A 0.000,B 0.000,C 90.000,E1 36.011} C_DIS
LIN {X 0.029,Y -550.812,Z 1056.995,A 0.000,B 0.000,C 90.000,E1 35.185} C_DIS
LIN {X 0.193,Y -546.892,Z 1056.991,A 0.000,B 0.000,C 90.000,E1 34.326} C_DIS
LIN {X 0.137,Y -543.425,Z 1056.987,A 0.000,B 0.000,C 90.000,E1 33.627} C_DIS
LIN {X 0.081,Y -537.456,Z 1056.981,A 0.000,B 0.000,C 90.000,E1 32.498} C_DIS
LIN {X 0.085,Y -534.245,Z 1056.977,A 0.000,B 0.000,C 90.000,E1 31.926} C_DIS
LIN {X 0.231,Y -530.835,Z 1056.974,A 0.000,B 0.000,C 90.000,E1 31.337} C_DIS
LIN {X -0.096,Y -527.245,Z 1056.971,A 0.000,B 0.000,C 90.000,E1 30.797} C_DIS
LIN {X 0.005,Y -523.337,Z 1056.968,A 0.000,B 0.000,C 90.000,E1 30.207} C_DIS
LIN {X 0.007,Y -517.120,Z 1056.963,A 0.000,B 0.000,C 90.000,E1 29.333} C_DIS
LIN {X -0.139,Y -511.453,Z 1056.959,A 0.000,B 0.000,C 90.000,E1 28.615} C_DIS
LIN {X -0.154,Y -506.600,Z 1056.956,A 0.000,B 0.000,C 90.000,E1 28.025} C_DIS
LIN {X 0.239,Y -501.324,Z 1056.952,A 0.000,B 0.000,C 90.000,E1 27.385} C_DIS
LIN {X 0.094,Y -494.737,Z 1056.948,A 0.000,B 0.000,C 90.000,E1 26.693} C_DIS
LIN {X 0.214,Y -487.833,Z 1056.944,A 0.000,B 0.000,C 90.000,E1 25.976} C_DIS
LIN {X 0.071,Y -479.301,Z 1056.940,A 0.000,B 0.000,C 90.000,E1 25.155} C_DIS
LIN {X 0.044,Y -470.542,Z 1056.935,A 0.000,B 0.000,C 90.000,E1 24.335} C_DIS
LIN {X -0.164,Y -464.494,Z 1056.932,A 0.000,B 0.000,C 90.000,E1 23.823} C_DIS
LIN {X 0.025,Y -455.408,Z 1056.928,A 0.000,B 0.000,C 90.000,E1 23.025} C_DIS
LIN {X -0.270,Y -444.868,Z 1056.923,A 0.000,B 0.000,C 90.000,E1 22.153} C_DIS
LIN {X -0.056,Y -425.611,Z 1056.913,A 0.000,B 0.000,C 90.000,E1 20.355} C_DIS
LIN {X -0.017,Y -413.016,Z 1056.906,A 0.000,B 0.000,C 90.000,E1 19.033} C_DIS
LIN {X 0.075,Y -402.300,Z 1056.899,A 0.000,B 0.000,C 90.000,E1 17.764} C_DIS
LIN {X -0.003,Y -397.611,Z 1056.895,A 0.000,B 0.000,C 90.000,E1 17.149} C_DIS
LIN {X -0.157,Y -394.968,Z 1056.893,A 0.000,B 0.000,C 90.000,E1 16.732} C_DIS
LIN {X -0.008,Y -393.425,Z 1056.891,A 0.000,B 0.000,C 90.000,E1 16.386} C_DIS
LIN {X -0.135,Y -392.414,Z 1056.889,A 0.000,B 0.000,C 90.000,E1 16.079} C_DIS
LIN {X -0.109,Y -391.693,Z 1056.886,A 0.000,B 0.000,C 90.000,E1 15.552} C_DIS
LIN {X -0.019,Y -391.654,Z 1056.882,A 0.000,B 0.000,C 90.000,E1 14.828} C_DIS
LIN {X -0.051,Y -393.995,Z 1056.871,A 0.000,B 0.000,C 90.000,E1 12.703} C_DIS
LIN {X 0.087,Y -399.910,Z 1056.849,A 0.000,B 0.000,C 90.000,E1 8.803} C_DIS
LIN {X -0.106,Y -407.722,Z 1056.828,A 0.000,B 0.000,C 90.000,E1 4.992} C_DIS
LIN {X -0.123,Y -409.256,Z 1056.824,A 0.000,B 0.000,C 90.000,E1 4.302} C_DIS
LIN {X -0.134,Y -411.781,Z 1056.819,A 0.000,B 0.000,C 90.000,E1 3.440} C_DIS
LIN {X -0.140,Y -412.570,Z 1056.818,A 0.000,B 0.000,C 90.000,E1 3.269} C_DIS
LIN {X -0.194,Y -415.134,Z 1056.816,A 0.000,B 0.000,C 90.000,E1 2.808} C_DIS
LIN {X -0.189,Y -417.687,Z 1056.814,A 0.000,B 0.000,C 90.000,E1 2.465} C_DIS
LIN {X 0.018,Y -422.742,Z 1056.811,A 0.000,B 0.000,C 90.000,E1 2.007} C_DIS
LIN {X -0.021,Y -438.647,Z 1056.805,A 0.000,B 0.000,C 90.000,E1 0.974} C_DIS
LIN {X 0.173,Y -457.311,Z 1056.799,A 0.000,B 0.000,C 90.000,E1 359.771} C_DIS
LIN {X 0.005,Y -475.379,Z 1056.793,A 0.000,B 0.000,C 90.000,E1 358.682} C_DIS
LIN {X 0.031,Y -486.646,Z 1056.789,A 0.000,B 0.000,C 90.000,E1 357.993} C_DIS
LIN {X 0.180,Y -496.302,Z 1056.786,A 0.000,B 0.000,C 90.000,E1 357.364} C_DIS
LIN {X 0.217,Y -503.952,Z 1056.783,A 0.000,B 0.000,C 90.000,E1 356.849} C_DIS
LIN {X 0.011,Y -511.583,Z 1056.780,A 0.000,B 0.000,C 90.000,E1 356.331} C_DIS
LIN {X 0.133,Y -517.491,Z 1056.777,A 0.000,B 0.000,C 90.000,E1 355.869} C_DIS
LIN {X -0.031,Y -523.347,Z 1056.775,A 0.000,B 0.000,C 90.000,E1 355.412} C_DIS
LIN {X -0.170,Y -528.867,Z 1056.772,A 0.000,B 0.000,C 90.000,E1 354.951} C_DIS
LIN {X -0.181,Y -534.485,Z 1056.769,A 0.000,B 0.000,C 90.000,E1 354.432} C_DIS
LIN {X 0.185,Y -540.774,Z 1056.765,A 0.000,B 0.000,C 90.000,E1 353.742} C_DIS
LIN {X 0.176,Y -546.859,Z 1056.762,A 0.000,B 0.000,C 90.000,E1 353.053} C_DIS
LIN {X -0.184,Y -551.324,Z 1056.758,A 0.000,B 0.000,C 90.000,E1 352.527} C_DIS
LIN {X -0.037,Y -555.462,Z 1056.755,A 0.000,B 0.000,C 90.000,E1 351.951} C_DIS
LIN {X -0.027,Y -560.048,Z 1056.751,A 0.000,B 0.000,C 90.000,E1 351.254} C_DIS
LIN {X -0.097,Y -564.926,Z 1056.747,A 0.000,B 0.000,C 90.000,E1 350.443} C_DIS
LIN {X 0.237,Y -567.921,Z 1056.744,A 0.000,B 0.000,C 90.000,E1 349.859} C_DIS
LIN {X 0.120,Y -572.084,Z 1056.739,A 0.000,B 0.000,C 90.000,E1 349.050} C_DIS
LIN {X -0.292,Y -575.276,Z 1056.735,A 0.000,B 0.000,C 90.000,E1 348.409} C_DIS
LIN {X -0.019,Y -579.988,Z 1056.729,A 0.000,B 0.000,C 90.000,E1 347.297} C_DIS
LIN {X -0.116,Y -584.331,Z 1056.724,A 0.000,B 0.000,C 90.000,E1 346.228} C_DIS
LIN {X 0.110,Y -589.514,Z 1056.716,A 0.000,B 0.000,C 90.000,E1 344.866} C_DIS
LIN {X 0.119,Y -595.354,Z 1056.707,A 0.000,B 0.000,C 90.000,E1 343.268} C_DIS
LIN {X -0.152,Y -598.965,Z 1056.701,A 0.000,B 0.000,C 90.000,E1 342.236} C_DIS
LIN {X 0.206,Y -602.357,Z 1056.695,A 0.000,B 0.000,C 90.000,E1 341.148} C_DIS
LIN {X 0.040,Y -605.421,Z 1056.690,A 0.000,B 0.000,C 90.000,E1 340.115} C_DIS
LIN {X -0.024,Y -607.581,Z 1056.685,A 0.000,B 0.000,C 90.000,E1 339.337} C_DIS
LIN {X 0.089,Y -610.341,Z 1056.679,A 0.000,B 0.000,C 90.000,E1 338.284} C_DIS
LIN {X 0.246,Y -612.832,Z 1056.674,A 0.000,B 0.000,C 90.000,E1 337.230} C_DIS
LIN {X -0.129,Y -615.151,Z 1056.668,A 0.000,B 0.000,C 90.000,E1 336.230} C_DIS
LIN {X 0.084,Y -617.133,Z 1056.662,A 0.000,B 0.000,C 90.000,E1 335.177} C_DIS
LIN {X 0.009,Y -619.281,Z 1056.655,A 0.000,B 0.000,C 90.000,E1 333.896} C_DIS
LIN {X -0.027,Y -621.103,Z 1056.648,A 0.000,B 0.000,C 90.000,E1 332.615} C_DIS
LIN {X 0.257,Y -622.719,Z 1056.641,A 0.000,B 0.000,C 90.000,E1 331.307} C_DIS
LIN {X -0.282,Y -623.815,Z 1056.635,A 0.000,B 0.000,C 90.000,E1 330.333} C_DIS
LIN {X 0.037,Y -624.629,Z 1056.629,A 0.000,B 0.000,C 90.000,E1 329.282} C_DIS
LIN {X 0.154,Y -625.222,Z 1056.624,A 0.000,B 0.000,C 90.000,E1 328.250} C_DIS
LIN {X -0.045,Y -625.696,Z 1056.618,A 0.000,B 0.000,C 90.000,E1 327.248} C_DIS
LIN {X 0.097,Y -625.802,Z 1056.612,A 0.000,B 0.000,C 90.000,E1 326.215} C_DIS
LIN {X -0.291,Y -625.714,Z 1056.605,A 0.000,B 0.000,C 90.000,E1 324.975} C_DIS
LIN {X 0.208,Y -625.515,Z 1056.600,A 0.000,B 0.000,C 90.000,E1 323.909} C_DIS
LIN {X -0.026,Y -625.036,Z 1056.590,A 0.000,B 0.000,C 90.000,E1 322.145} C_DIS
LIN {X 0.193,Y -624.577,Z 1056.577,A 0.000,B 0.000,C 90.000,E1 319.828} C_DIS
LIN {X 0.025,Y -624.462,Z 1056.570,A 0.000,B 0.000,C 90.000,E1 318.566} C_DIS
LIN {X -0.203,Y -624.205,Z 1056.563,A 0.000,B 0.000,C 90.000,E1 317.310} C_DIS
LIN {X 0.183,Y -623.926,Z 1056.553,A 0.000,B 0.000,C 90.000,E1 315.486} C_DIS
LIN {X 0.112,Y -623.660,Z 1056.543,A 0.000,B 0.000,C 90.000,E1 313.704} C_DIS
LIN {X 0.154,Y -623.564,Z 1056.539,A 0.000,B 0.000,C 90.000,E1 312.933} C_DIS
LIN {X 0.058,Y -623.286,Z 1056.533,A 0.000,B 0.000,C 90.000,E1 311.919} C_DIS
LIN {X -0.093,Y -622.616,Z 1056.522,A 0.000,B 0.000,C 90.000,E1 309.886} C_DIS
LIN {X 0.262,Y -622.300,Z 1056.516,A 0.000,B 0.000,C 90.000,E1 308.830} C_DIS
LIN {X 0.167,Y -621.928,Z 1056.505,A 0.000,B 0.000,C 90.000,E1 306.790} C_DIS
LIN {X 0.070,Y -621.752,Z 1056.497,A 0.000,B 0.000,C 90.000,E1 305.518} C_DIS
LIN {X 0.267,Y -621.834,Z 1056.487,A 0.000,B 0.000,C 90.000,E1 303.706} C_DIS
LIN {X 0.108,Y -622.180,Z 1056.476,A 0.000,B 0.000,C 90.000,E1 301.671} C_DIS
LIN {X 0.175,Y -622.509,Z 1056.468,A 0.000,B 0.000,C 90.000,E1 300.129} C_DIS
LIN {X 0.172,Y -622.670,Z 1056.465,A 0.000,B 0.000,C 90.000,E1 299.617} C_DIS
LIN {X -0.064,Y -622.996,Z 1056.458,A 0.000,B 0.000,C 90.000,E1 298.359} C_DIS
LIN {X -0.056,Y -623.121,Z 1056.455,A 0.000,B 0.000,C 90.000,E1 297.847} C_DIS
LIN {X -0.036,Y -622.890,Z 1056.449,A 0.000,B 0.000,C 90.000,E1 296.821} C_DIS
LIN {X -0.030,Y -622.977,Z 1056.448,A 0.000,B 0.000,C 90.000,E1 296.565} C_DIS
LIN {X -0.010,Y -622.399,Z 1056.442,A 0.000,B 0.000,C 90.000,E1 295.540} C_DIS
LIN {X -0.008,Y -622.446,Z 1056.441,A 0.000,B 0.000,C 90.000,E1 295.283} C_DIS
LIN {X -0.007,Y -621.417,Z 1056.435,A 0.000,B 0.000,C 90.000,E1 294.259} C_DIS
LIN {X -0.267,Y -620.803,Z 1056.432,A 0.000,B 0.000,C 90.000,E1 293.770} C_DIS
LIN {X -0.272,Y -620.548,Z 1056.431,A 0.000,B 0.000,C 90.000,E1 293.515} C_DIS
LIN {X 0.016,Y -618.641,Z 1056.425,A 0.000,B 0.000,C 90.000,E1 292.461} C_DIS
LIN {X -0.020,Y -617.419,Z 1056.422,A 0.000,B 0.000,C 90.000,E1 291.950} C_DIS
LIN {X -0.271,Y -616.666,Z 1056.421,A 0.000,B 0.000,C 90.000,E1 291.716} C_DIS
LIN {X 0.025,Y -614.784,Z 1056.418,A 0.000,B 0.000,C 90.000,E1 291.173} C_DIS
LIN {X -0.047,Y -611.774,Z 1056.415,A 0.000,B 0.000,C 90.000,E1 290.663} C_DIS
LIN {X -0.285,Y -610.786,Z 1056.414,A 0.000,B 0.000,C 90.000,E1 290.556} C_DIS
LIN {X 0.227,Y -607.286,Z 1056.412,A 0.000,B 0.000,C 90.000,E1 290.120} C_DIS
LIN {X 0.195,Y -605.842,Z 1056.411,A 0.000,B 0.000,C 90.000,E1 289.993} C_DIS
LIN {X -0.042,Y -604.188,Z 1056.411,A 0.000,B 0.000,C 90.000,E1 289.885} C_DIS
LIN {X -0.279,Y -602.554,Z 1056.410,A 0.000,B 0.000,C 90.000,E1 289.758} C_DIS
LIN {X -0.219,Y -600.987,Z 1056.409,A 0.000,B 0.000,C 90.000,E1 289.631} C_DIS
LIN {X 0.159,Y -596.977,Z 1056.408,A 0.000,B 0.000,C 90.000,E1 289.396} C_DIS
LIN {X 0.009,Y -594.729,Z 1056.407,A 0.000,B 0.000,C 90.000,E1 289.214} C_DIS
LIN {X 0.099,Y -592.707,Z 1056.406,A 0.000,B 0.000,C 90.000,E1 289.087} C_DIS
LIN {X 0.222,Y -585.796,Z 1056.404,A 0.000,B 0.000,C 90.000,E1 288.725} C_DIS
LIN {X -0.170,Y -578.593,Z 1056.403,A 0.000,B 0.000,C 90.000,E1 288.598} C_DIS
LIN {X 0.176,Y -573.942,Z 1056.402,A 0.000,B 0.000,C 90.000,E1 288.362} C_DIS
LIN {X -0.043,Y -564.984,Z 1056.401,A 0.000,B 0.000,C 90.000,E1 288.127} C_DIS
LIN {X 0.200,Y -562.734,Z 1056.401,A 0.000,B 0.000,C 90.000,E1 288.055} C_DIS
LIN {X 0.265,Y -557.831,Z 1056.400,A 0.000,B 0.000,C 90.000,E1 288.000} C_DIS
LIN {X -0.027,Y -553.032,Z 1056.400,A 0.000,B 0.000,C 90.000,E1 288.000} C_DIS
LIN {X 0.143,Y -549.939,Z 1056.399,A 0.000,B 0.000,C 90.000,E1 287.819} C_DIS
LIN {X 0.245,Y -547.149,Z 1056.398,A 0.000,B 0.000,C 90.000,E1 287.638} C_DIS
LIN {X 0.216,Y -547.139,Z 1056.398,A 0.000,B 0.000,C 90.000,E1 287.638} C_DIS
LIN {X 0.050,Y -546.254,Z 1056.396,A 0.000,B 0.000,C 90.000,E1 287.347} C_DIS
LIN {X -0.130,Y -545.657,Z 1056.393,A 0.000,B 0.000,C 90.000,E1 286.804} C_DIS
LIN {X -0.041,Y -544.918,Z 1056.381,A 0.000,B 0.000,C 90.000,E1 284.537} C_DIS
LIN {X -0.086,Y -544.559,Z 1056.375,A 0.000,B 0.000,C 90.000,E1 283.411} C_DIS
LIN {X -0.175,Y -543.832,Z 1056.367,A 0.000,B 0.000,C 90.000,E1 282.007} C_DIS
LIN {X -0.189,Y -542.828,Z 1056.357,A 0.000,B 0.000,C 90.000,E1 280.310} C_DIS
LIN {X 0.129,Y -542.004,Z 1056.349,A 0.000,B 0.000,C 90.000,E1 278.859} C_DIS
LIN {X -0.107,Y -540.934,Z 1056.340,A 0.000,B 0.000,C 90.000,E1 277.182} C_DIS
LIN {X 0.040,Y -540.291,Z 1056.334,A 0.000,B 0.000,C 90.000,E1 276.030} C_DIS
LIN {X 0.243,Y -539.254,Z 1056.324,A 0.000,B 0.000,C 90.000,E1 274.302} C_DIS
LIN {X -0.173,Y -538.448,Z 1056.316,A 0.000,B 0.000,C 90.000,E1 272.922} C_DIS
LIN {X -0.089,Y -537.532,Z 1056.307,A 0.000,B 0.000,C 90.000,E1 271.203} C_DIS
LIN {X -0.033,Y -536.456,Z 1056.297,A 0.000,B 0.000,C 90.000,E1 269.484} C_DIS
LIN {X 0.011,Y -535.437,Z 1056.288,A 0.000,B 0.000,C 90.000,E1 267.764} C_DIS
LIN {X 0.033,Y -534.493,Z 1056.280,A 0.000,B 0.000,C 90.000,E1 266.331} C_DIS
LIN {X 0.070,Y -533.472,Z 1056.272,A 0.000,B 0.000,C 90.000,E1 264.894} C_DIS
LIN {X 0.081,Y -532.368,Z 1056.264,A 0.000,B 0.000,C 90.000,E1 263.457} C_DIS
LIN {X 0.160,Y -531.261,Z 1056.257,A 0.000,B 0.000,C 90.000,E1 262.299} C_DIS
LIN {X -0.247,Y -528.822,Z 1056.245,A 0.000,B 0.000,C 90.000,E1 260.038} C_DIS
LIN {X -0.124,Y -527.569,Z 1056.238,A 0.000,B 0.000,C 90.000,E1 258.870} C_DIS
LIN {X 0.026,Y -525.648,Z 1056.229,A 0.000,B 0.000,C 90.000,E1 257.117} C_DIS
LIN {X -0.126,Y -523.504,Z 1056.217,A 0.000,B 0.000,C 90.000,E1 255.102} C_DIS
LIN {X 0.177,Y -522.012,Z 1056.209,A 0.000,B 0.000,C 90.000,E1 253.614} C_DIS
LIN {X -0.198,Y -520.804,Z 1056.203,A 0.000,B 0.000,C 90.000,E1 252.489} C_DIS
LIN {X -0.158,Y -518.827,Z 1056.193,A 0.000,B 0.000,C 90.000,E1 250.732} C_DIS
LIN {X 0.154,Y -516.368,Z 1056.182,A 0.000,B 0.000,C 90.000,E1 248.646} C_DIS
LIN {X 0.141,Y -514.420,Z 1056.173,A 0.000,B 0.000,C 90.000,E1 247.177} C_DIS
LIN {X 0.160,Y -512.733,Z 1056.167,A 0.000,B 0.000,C 90.000,E1 245.997} C_DIS
LIN {X -0.100,Y -510.993,Z 1056.160,A 0.000,B 0.000,C 90.000,E1 244.845} C_DIS
LIN {X -0.276,Y -508.563,Z 1056.152,A 0.000,B 0.000,C 90.000,E1 243.384} C_DIS
LIN {X 0.097,Y -506.636,Z 1056.145,A 0.000,B 0.000,C 90.000,E1 242.153} C_DIS
LIN {X 0.063,Y -504.116,Z 1056.137,A 0.000,B 0.000,C 90.000,E1 240.667} C_DIS
LIN {X -0.212,Y -501.347,Z 1056.129,A 0.000,B 0.000,C 90.000,E1 239.203} C_DIS
LIN {X 0.016,Y -498.048,Z 1056.119,A 0.000,B 0.000,C 90.000,E1 237.375} C_DIS
LIN {X -0.109,Y -495.124,Z 1056.110,A 0.000,B 0.000,C 90.000,E1 235.881} C_DIS
LIN {X -0.019,Y -492.142,Z 1056.102,A 0.000,B 0.000,C 90.000,E1 234.356} C_DIS
LIN {X 0.059,Y -489.371,Z 1056.095,A 0.000,B 0.000,C 90.000,E1 233.130} C_DIS
LIN {X 0.064,Y -485.122,Z 1056.085,A 0.000,B 0.000,C 90.000,E1 231.295} C_DIS
LIN {X -0.027,Y -480.934,Z 1056.075,A 0.000,B 0.000,C 90.000,E1 229.461} C_DIS
LIN {X -0.160,Y -476.382,Z 1056.063,A 0.000,B 0.000,C 90.000,E1 227.310} C_DIS
LIN {X -0.164,Y -474.530,Z 1056.058,A 0.000,B 0.000,C 90.000,E1 226.377} C_DIS
LIN {X -0.006,Y -471.483,Z 1056.049,A 0.000,B 0.000,C 90.000,E1 224.798} C_DIS
LIN {X -0.152,Y -467.695,Z 1056.038,A 0.000,B 0.000,C 90.000,E1 222.933} C_DIS
LIN {X -0.023,Y -463.919,Z 1056.028,A 0.000,B 0.000,C 90.000,E1 221.024} C_DIS
LIN {X -0.169,Y -461.903,Z 1056.023,A 0.000,B 0.000,C 90.000,E1 220.092} C_DIS
LIN {X 0.138,Y -458.613,Z 1056.014,A 0.000,B 0.000,C 90.000,E1 218.463} C_DIS
LIN {X -0.178,Y -454.730,Z 1056.003,A 0.000,B 0.000,C 90.000,E1 216.583} C_DIS
LIN {X 0.062,Y -451.440,Z 1055.994,A 0.000,B 0.000,C 90.000,E1 214.945} C_DIS
LIN {X 0.184,Y -446.002,Z 1055.980,A 0.000,B 0.000,C 90.000,E1 212.339} C_DIS
LIN {X 0.060,Y -443.254,Z 1055.973,A 0.000,B 0.000,C 90.000,E1 211.052} C_DIS
LIN {X 0.138,Y -439.068,Z 1055.962,A 0.000,B 0.000,C 90.000,E1 209.077} C_DIS
LIN {X 0.136,Y -433.565,Z 1055.947,A 0.000,B 0.000,C 90.000,E1 206.437} C_DIS
LIN {X 0.167,Y -430.164,Z 1055.938,A 0.000,B 0.000,C 90.000,E1 204.771} C_DIS
LIN {X 0.083,Y -424.614,Z 1055.921,A 0.000,B 0.000,C 90.000,E1 201.770} C_DIS
LIN {X 0.132,Y -420.144,Z 1055.904,A 0.000,B 0.000,C 90.000,E1 198.725} C_DIS
LIN {X 0.243,Y -419.071,Z 1055.899,A 0.000,B 0.000,C 90.000,E1 197.692} C_DIS
LIN {X 0.214,Y -418.366,Z 1055.893,A 0.000,B 0.000,C 90.000,E1 196.677} C_DIS
LIN {X 0.177,Y -417.950,Z 1055.887,A 0.000,B 0.000,C 90.000,E1 195.662} C_DIS
LIN {X -0.179,Y -417.947,Z 1055.885,A 0.000,B 0.000,C 90.000,E1 195.371} C_DIS
LIN {X 0.027,Y -418.295,Z 1055.881,A 0.000,B 0.000,C 90.000,E1 194.662} C_DIS
LIN {X -0.169,Y -418.951,Z 1055.878,A 0.000,B 0.000,C 90.000,E1 194.008} C_DIS
LIN {X 0.045,Y -420.170,Z 1055.874,A 0.000,B 0.000,C 90.000,E1 193.300} C_DIS
LIN {X -0.156,Y -422.619,Z 1055.869,A 0.000,B 0.000,C 90.000,E1 192.479} C_DIS
LIN {X 0.172,Y -426.167,Z 1055.865,A 0.000,B 0.000,C 90.000,E1 191.591} C_DIS
LIN {X 0.155,Y -431.458,Z 1055.859,A 0.000,B 0.000,C 90.000,E1 190.602} C_DIS
LIN {X -0.203,Y -439.483,Z 1055.852,A 0.000,B 0.000,C 90.000,E1 189.321} C_DIS
LIN {X 0.179,Y -451.257,Z 1055.842,A 0.000,B 0.000,C 90.000,E1 187.473} C_DIS
LIN {X -0.027,Y -458.795,Z 1055.835,A 0.000,B 0.000,C 90.000,E1 186.372} C_DIS
LIN {X 0.236,Y -465.038,Z 1055.830,A 0.000,B 0.000,C 90.000,E1 185.391} C_DIS
LIN {X -0.117,Y -470.090,Z 1055.826,A 0.000,B 0.000,C 90.000,E1 184.645} C_DIS
LIN {X -0.174,Y -476.864,Z 1055.820,A 0.000,B 0.000,C 90.000,E1 183.555} C_DIS
LIN {X 0.011,Y -484.451,Z 1055.813,A 0.000,B 0.000,C 90.000,E1 182.293} C_DIS
LIN {X -0.013,Y -489.937,Z 1055.808,A 0.000,B 0.000,C 90.000,E1 181.375} C_DIS
LIN {X 0.229,Y -498.913,Z 1055.799,A 0.000,B 0.000,C 90.000,E1 179.828} C_DIS
LIN {X 0.139,Y -507.413,Z 1055.791,A 0.000,B 0.000,C 90.000,E1 178.339} C_DIS
LIN {X -0.219,Y -514.103,Z 1055.784,A 0.000,B 0.000,C 90.000,E1 177.192} C_DIS
LIN {X -0.045,Y -523.869,Z 1055.775,A 0.000,B 0.000,C 90.000,E1 175.412} C_DIS
LIN {X -0.106,Y -531.816,Z 1055.766,A 0.000,B 0.000,C 90.000,E1 173.970} C_DIS
LIN {X 0.192,Y -538.784,Z 1055.759,A 0.000,B 0.000,C 90.000,E1 172.648} C_DIS
LIN {X -0.056,Y -546.492,Z 1055.751,A 0.000,B 0.000,C 90.000,E1 171.254} C_DIS
LIN {X -0.161,Y -553.988,Z 1055.744,A 0.000,B 0.000,C 90.000,E1 169.859} C_DIS
LIN {X 0.113,Y -560.557,Z 1055.737,A 0.000,B 0.000,C 90.000,E1 168.578} C_DIS
LIN {X 0.107,Y -568.229,Z 1055.728,A 0.000,B 0.000,C 90.000,E1 167.061} C_DIS
LIN {X -0.137,Y -573.615,Z 1055.722,A 0.000,B 0.000,C 90.000,E1 165.992} C_DIS
LIN {X 0.010,Y -579.317,Z 1055.715,A 0.000,B 0.000,C 90.000,E1 164.755} C_DIS
LIN {X 0.258,Y -582.994,Z 1055.711,A 0.000,B 0.000,C 90.000,E1 163.921} C_DIS
LIN {X -0.018,Y -586.559,Z 1055.706,A 0.000,B 0.000,C 90.000,E1 163.142} C_DIS
LIN {X 0.163,Y -591.092,Z 1055.700,A 0.000,B 0.000,C 90.000,E1 162.054} C_DIS
LIN {X -0.035,Y -594.224,Z 1055.696,A 0.000,B 0.000,C 90.000,E1 161.275} C_DIS
LIN {X 0.251,Y -598.235,Z 1055.690,A 0.000,B 0.000,C 90.000,E1 160.188} C_DIS
LIN {X 0.023,Y -602.064,Z 1055.684,A 0.000,B 0.000,C 90.000,E1 159.156} C_DIS
LIN {X -0.006,Y -606.487,Z 1055.677,A 0.000,B 0.000,C 90.000,E1 157.847} C_DIS
LIN {X 0.149,Y -608.941,Z 1055.673,A 0.000,B 0.000,C 90.000,E1 157.050} C_DIS
LIN {X 0.244,Y -612.888,Z 1055.665,A 0.000,B 0.000,C 90.000,E1 155.741} C_DIS
LIN {X 0.082,Y -617.189,Z 1055.657,A 0.000,B 0.000,C 90.000,E1 154.204} C_DIS
LIN {X 0.024,Y -620.568,Z 1055.650,A 0.000,B 0.000,C 90.000,E1 152.922} C_DIS
LIN {X 0.015,Y -623.718,Z 1055.642,A 0.000,B 0.000,C 90.000,E1 151.641} C_DIS
LIN {X 0.341,Y -626.220,Z 1055.637,A 0.000,B 0.000,C 90.000,E1 150.589} C_DIS
LIN {X 0.176,Y -629.275,Z 1055.630,A 0.000,B 0.000,C 90.000,E1 149.331} C_DIS
LIN {X 0.410,Y -632.683,Z 1055.621,A 0.000,B 0.000,C 90.000,E1 147.788} C_DIS
LIN {X -0.335,Y -636.568,Z 1055.611,A 0.000,B 0.000,C 90.000,E1 146.087} C_DIS
LIN {X -0.152,Y -639.827,Z 1055.603,A 0.000,B 0.000,C 90.000,E1 144.562} C_DIS
LIN {X 0.363,Y -643.587,Z 1055.593,A 0.000,B 0.000,C 90.000,E1 142.763} C_DIS
LIN {X 0.062,Y -647.334,Z 1055.584,A 0.000,B 0.000,C 90.000,E1 141.045} C_DIS
LIN {X 0.218,Y -650.545,Z 1055.575,A 0.000,B 0.000,C 90.000,E1 139.542} C_DIS
LIN {X -0.094,Y -654.310,Z 1055.566,A 0.000,B 0.000,C 90.000,E1 137.838} C_DIS
LIN {X -0.287,Y -657.626,Z 1055.558,A 0.000,B 0.000,C 90.000,E1 136.377} C_DIS
LIN {X -0.046,Y -665.144,Z 1055.541,A 0.000,B 0.000,C 90.000,E1 133.419} C_DIS
LIN {X -0.064,Y -669.039,Z 1055.533,A 0.000,B 0.000,C 90.000,E1 131.962} C_DIS
LIN {X 0.107,Y -673.570,Z 1055.524,A 0.000,B 0.000,C 90.000,E1 130.253} C_DIS
LIN {X -0.147,Y -677.449,Z 1055.516,A 0.000,B 0.000,C 90.000,E1 128.830} C_DIS
LIN {X 0.173,Y -680.553,Z 1055.509,A 0.000,B 0.000,C 90.000,E1 127.604} C_DIS
LIN {X 0.187,Y -684.789,Z 1055.500,A 0.000,B 0.000,C 90.000,E1 125.931} C_DIS
LIN {X 0.218,Y -687.791,Z 1055.493,A 0.000,B 0.000,C 90.000,E1 124.739} C_DIS
LIN {X -0.451,Y -691.268,Z 1055.485,A 0.000,B 0.000,C 90.000,E1 123.372} C_DIS
LIN {X -0.346,Y -693.589,Z 1055.480,A 0.000,B 0.000,C 90.000,E1 122.418} C_DIS
LIN {X 0.032,Y -696.284,Z 1055.474,A 0.000,B 0.000,C 90.000,E1 121.209} C_DIS
LIN {X -0.059,Y -697.832,Z 1055.469,A 0.000,B 0.000,C 90.000,E1 120.512} C_DIS
LIN {X 0.107,Y -699.176,Z 1055.466,A 0.000,B 0.000,C 90.000,E1 119.795} C_DIS
LIN {X 0.290,Y -700.306,Z 1055.462,A 0.000,B 0.000,C 90.000,E1 119.077} C_DIS
LIN {X 0.216,Y -700.889,Z 1055.459,A 0.000,B 0.000,C 90.000,E1 118.615} C_DIS
LIN {X -0.114,Y -703.056,Z 1055.447,A 0.000,B 0.000,C 90.000,E1 116.539} C_DIS
LIN {X 0.071,Y -703.936,Z 1055.442,A 0.000,B 0.000,C 90.000,E1 115.591} C_DIS
LIN {X -0.012,Y -704.390,Z 1055.438,A 0.000,B 0.000,C 90.000,E1 114.899} C_DIS
LIN {X 0.273,Y -704.502,Z 1055.437,A 0.000,B 0.000,C 90.000,E1 114.643} C_DIS
LIN {X -0.089,Y -704.270,Z 1055.434,A 0.000,B 0.000,C 90.000,E1 114.207} C_DIS
LIN {X 0.194,Y -703.990,Z 1055.433,A 0.000,B 0.000,C 90.000,E1 113.951} C_DIS
LIN {X -0.170,Y -702.735,Z 1055.431,A 0.000,B 0.000,C 90.000,E1 113.515} C_DIS
LIN {X 0.108,Y -701.680,Z 1055.429,A 0.000,B 0.000,C 90.000,E1 113.259} C_DIS
LIN {X -0.219,Y -698.486,Z 1055.427,A 0.000,B 0.000,C 90.000,E1 112.823} C_DIS
LIN {X -0.088,Y -697.411,Z 1055.426,A 0.000,B 0.000,C 90.000,E1 112.695} C_DIS
LIN {X -0.226,Y -695.780,Z 1055.425,A 0.000,B 0.000,C 90.000,E1 112.589} C_DIS
LIN {X 0.195,Y -688.419,Z 1055.423,A 0.000,B 0.000,C 90.000,E1 112.206} C_DIS
LIN {X -0.071,Y -686.456,Z 1055.423,A 0.000,B 0.000,C 90.000,E1 112.153} C_DIS
LIN {X -0.078,Y -683.357,Z 1055.423,A 0.000,B 0.000,C 90.000,E1 112.078} C_DIS
LIN {X 0.097,Y -676.051,Z 1055.422,A 0.000,B 0.000,C 90.000,E1 111.972} C_DIS
LIN {X 0.029,Y -609.442,Z 1055.422,A 0.000,B 0.000,C 90.000,E1 111.972} C_DIS
LIN {X -0.281,Y -605.017,Z 1055.421,A 0.000,B 0.000,C 90.000,E1 111.844} C_DIS
LIN {X 0.058,Y -602.776,Z 1055.421,A 0.000,B 0.000,C 90.000,E1 111.716} C_DIS
LIN {X 0.094,Y -596.289,Z 1055.419,A 0.000,B 0.000,C 90.000,E1 111.354} C_DIS
LIN {X 0.102,Y -591.025,Z 1055.417,A 0.000,B 0.000,C 90.000,E1 110.972} C_DIS
LIN {X 0.107,Y -578.489,Z 1055.411,A 0.000,B 0.000,C 90.000,E1 109.939} C_DIS
LIN {X 0.255,Y -574.110,Z 1055.409,A 0.000,B 0.000,C 90.000,E1 109.577} C_DIS
LIN {X -0.021,Y -569.632,Z 1055.407,A 0.000,B 0.000,C 90.000,E1 109.268} C_DIS
LIN {X -0.146,Y -561.149,Z 1055.404,A 0.000,B 0.000,C 90.000,E1 108.779} C_DIS
LIN {X 0.161,Y -553.485,Z 1055.402,A 0.000,B 0.000,C 90.000,E1 108.308} C_DIS
LIN {X 0.171,Y -549.636,Z 1055.401,A 0.000,B 0.000,C 90.000,E1 108.055} C_DIS
LIN {X 0.260,Y -548.179,Z 1055.400,A 0.000,B 0.000,C 90.000,E1 107.873} C_DIS
LIN {X 0.278,Y -547.772,Z 1055.399,A 0.000,B 0.000,C 90.000,E1 107.819} C_DIS
LIN {X 0.236,Y -547.739,Z 1055.399,A 0.000,B 0.000,C 90.000,E1 107.819} C_DIS
LIN {X -0.324,Y -547.231,Z 1055.398,A 0.000,B 0.000,C 90.000,E1 107.583} C_DIS
LIN {X 0.113,Y -548.466,Z 1055.386,A 0.000,B 0.000,C 90.000,E1 105.426} C_DIS
LIN {X 0.139,Y -549.938,Z 1055.373,A 0.000,B 0.000,C 90.000,E1 103.175} C_DIS
LIN {X -0.044,Y -551.853,Z 1055.361,A 0.000,B 0.000,C 90.000,E1 100.950} C_DIS
LIN {X 0.183,Y -554.236,Z 1055.348,A 0.000,B 0.000,C 90.000,E1 98.690} C_DIS
LIN {X 0.051,Y -555.492,Z 1055.342,A 0.000,B 0.000,C 90.000,E1 97.587} C_DIS
LIN {X -0.009,Y -557.140,Z 1055.334,A 0.000,B 0.000,C 90.000,E1 96.201} C_DIS
LIN {X -0.176,Y -558.286,Z 1055.328,A 0.000,B 0.000,C 90.000,E1 95.106} C_DIS
LIN {X 0.104,Y -558.945,Z 1055.324,A 0.000,B 0.000,C 90.000,E1 94.245} C_DIS
LIN {X -0.080,Y -559.721,Z 1055.318,A 0.000,B 0.000,C 90.000,E1 93.154} C_DIS
LIN {X -0.251,Y -560.331,Z 1055.311,A 0.000,B 0.000,C 90.000,E1 92.064} C_DIS
LIN {X -0.135,Y -561.086,Z 1055.301,A 0.000,B 0.000,C 90.000,E1 90.115} C_DIS
LIN {X -0.212,Y -561.517,Z 1055.293,A 0.000,B 0.000,C 90.000,E1 88.740} C_DIS
LIN {X -0.173,Y -562.040,Z 1055.284,A 0.000,B 0.000,C 90.000,E1 87.078} C_DIS
LIN {X -0.092,Y -562.747,Z 1055.275,A 0.000,B 0.000,C 90.000,E1 85.412} C_DIS
LIN {X -0.094,Y -563.128,Z 1055.267,A 0.000,B 0.000,C 90.000,E1 84.033} C_DIS
LIN {X 0.280,Y -563.603,Z 1055.256,A 0.000,B 0.000,C 90.000,E1 82.064} C_DIS
LIN {X -0.203,Y -564.061,Z 1055.248,A 0.000,B 0.000,C 90.000,E1 80.735} C_DIS
LIN {X 0.069,Y -565.053,Z 1055.235,A 0.000,B 0.000,C 90.000,E1 78.229} C_DIS
LIN {X -0.196,Y -565.770,Z 1055.227,A 0.000,B 0.000,C 90.000,E1 76.881} C_DIS
LIN {X -0.213,Y -567.094,Z 1055.215,A 0.000,B 0.000,C 90.000,E1 74.685} C_DIS
LIN {X 0.019,Y -568.314,Z 1055.206,A 0.000,B 0.000,C 90.000,E1 73.015} C_DIS
LIN {X 0.066,Y -569.861,Z 1055.195,A 0.000,B 0.000,C 90.000,E1 71.094} C_DIS
LIN {X 0.167,Y -571.297,Z 1055.186,A 0.000,B 0.000,C 90.000,E1 69.444} C_DIS
LIN {X 0.125,Y -572.747,Z 1055.175,A 0.000,B 0.000,C 90.000,E1 67.539} C_DIS
LIN {X -0.199,Y -574.052,Z 1055.165,A 0.000,B 0.000,C 90.000,E1 65.665} C_DIS
LIN {X -0.258,Y -575.108,Z 1055.154,A 0.000,B 0.000,C 90.000,E1 63.768} C_DIS
LIN {X -0.099,Y -575.702,Z 1055.148,A 0.000,B 0.000,C 90.000,E1 62.666} C_DIS
LIN {X -0.230,Y -576.542,Z 1055.139,A 0.000,B 0.000,C 90.000,E1 61.051} C_DIS
LIN {X -0.075,Y -577.241,Z 1055.130,A 0.000,B 0.000,C 90.000,E1 59.410} C_DIS
LIN {X -0.098,Y -577.672,Z 1055.124,A 0.000,B 0.000,C 90.000,E1 58.329} C_DIS
LIN {X -0.114,Y -578.117,Z 1055.118,A 0.000,B 0.000,C 90.000,E1 57.248} C_DIS
LIN {X 0.028,Y -578.579,Z 1055.110,A 0.000,B 0.000,C 90.000,E1 55.881} C_DIS
LIN {X 0.020,Y -579.121,Z 1055.100,A 0.000,B 0.000,C 90.000,E1 53.989} C_DIS
LIN {X -0.134,Y -579.125,Z 1055.094,A 0.000,B 0.000,C 90.000,E1 52.924} C_DIS
LIN {X 0.229,Y -579.041,Z 1055.087,A 0.000,B 0.000,C 90.000,E1 51.537} C_DIS
LIN {X -0.019,Y -578.670,Z 1055.080,A 0.000,B 0.000,C 90.000,E1 50.481} C_DIS
LIN {X 0.175,Y -578.211,Z 1055.074,A 0.000,B 0.000,C 90.000,E1 49.380} C_DIS
LIN {X 0.064,Y -577.544,Z 1055.067,A 0.000,B 0.000,C 90.000,E1 48.038} C_DIS
LIN {X -0.247,Y -576.825,Z 1055.061,A 0.000,B 0.000,C 90.000,E1 46.986} C_DIS
LIN {X -0.139,Y -575.886,Z 1055.055,A 0.000,B 0.000,C 90.000,E1 45.891} C_DIS
LIN {X -0.175,Y -575.022,Z 1055.050,A 0.000,B 0.000,C 90.000,E1 45.081} C_DIS
LIN {X 0.303,Y -573.644,Z 1055.044,A 0.000,B 0.000,C 90.000,E1 43.947} C_DIS
LIN {X -0.057,Y -571.975,Z 1055.038,A 0.000,B 0.000,C 90.000,E1 42.894} C_DIS
LIN {X 0.398,Y -570.192,Z 1055.032,A 0.000,B 0.000,C 90.000,E1 41.757} C_DIS
LIN {X -0.092,Y -568.638,Z 1055.028,A 0.000,B 0.000,C 90.000,E1 40.987} C_DIS
LIN {X -0.166,Y -566.770,Z 1055.023,A 0.000,B 0.000,C 90.000,E1 40.172} C_DIS
LIN {X -0.368,Y -565.480,Z 1055.020,A 0.000,B 0.000,C 90.000,E1 39.644} C_DIS
LIN {X 0.320,Y -563.215,Z 1055.016,A 0.000,B 0.000,C 90.000,E1 38.749} C_DIS
LIN {X 0.088,Y -561.618,Z 1055.012,A 0.000,B 0.000,C 90.000,E1 38.222} C_DIS
LIN {X 0.040,Y -558.872,Z 1055.008,A 0.000,B 0.000,C 90.000,E1 37.397} C_DIS
LIN {X -0.137,Y -555.802,Z 1055.003,A 0.000,B 0.000,C 90.000,E1 36.583} C_DIS
LIN {X 0.094,Y -552.586,Z 1054.999,A 0.000,B 0.000,C 90.000,E1 35.724} C_DIS
LIN {X -0.037,Y -548.803,Z 1054.994,A 0.000,B 0.000,C 90.000,E1 34.898} C_DIS
LIN {X -0.070,Y -545.426,Z 1054.990,A 0.000,B 0.000,C 90.000,E1 34.199} C_DIS
LIN {X -0.165,Y -543.344,Z 1054.988,A 0.000,B 0.000,C 90.000,E1 33.785} C_DIS
LIN {X -0.065,Y -536.517,Z 1054.981,A 0.000,B 0.000,C 90.000,E1 32.498} C_DIS
LIN {X -0.068,Y -533.296,Z 1054.977,A 0.000,B 0.000,C 90.000,E1 31.926} C_DIS
LIN {X -0.076,Y -528.972,Z 1054.973,A 0.000,B 0.000,C 90.000,E1 31.209} C_DIS
LIN {X 0.307,Y -525.245,Z 1054.970,A 0.000,B 0.000,C 90.000,E1 30.590} C_DIS
LIN {X 0.227,Y -520.251,Z 1054.966,A 0.000,B 0.000,C 90.000,E1 29.873} C_DIS
LIN {X -0.061,Y -513.786,Z 1054.961,A 0.000,B 0.000,C 90.000,E1 29.027} C_DIS
LIN {X 0.121,Y -510.312,Z 1054.959,A 0.000,B 0.000,C 90.000,E1 28.565} C_DIS
LIN {X 0.162,Y -505.466,Z 1054.956,A 0.000,B 0.000,C 90.000,E1 27.975} C_DIS
LIN {X -0.046,Y -497.645,Z 1054.951,A 0.000,B 0.000,C 90.000,E1 27.129} C_DIS
LIN {X -0.073,Y -490.709,Z 1054.947,A 0.000,B 0.000,C 90.000,E1 26.411} C_DIS
LIN {X 0.119,Y -480.881,Z 1054.941,A 0.000,B 0.000,C 90.000,E1 25.412} C_DIS
LIN {X 0.074,Y -469.363,Z 1054.935,A 0.000,B 0.000,C 90.000,E1 24.335} C_DIS
LIN {X 0.059,Y -462.038,Z 1054.932,A 0.000,B 0.000,C 90.000,E1 23.695} C_DIS
LIN {X 0.182,Y -448.431,Z 1054.925,A 0.000,B 0.000,C 90.000,E1 22.514} C_DIS
LIN {X -0.023,Y -427.612,Z 1054.915,A 0.000,B 0.000,C 90.000,E1 20.663} C_DIS
LIN {X -0.134,Y -416.109,Z 1054.908,A 0.000,B 0.000,C 90.000,E1 19.504} C_DIS
LIN {X 0.123,Y -407.868,Z 1054.903,A 0.000,B 0.000,C 90.000,E1 18.544} C_DIS
LIN {X -0.013,Y -399.869,Z 1054.898,A 0.000,B 0.000,C 90.000,E1 17.583} C_DIS
LIN {X -0.028,Y -396.408,Z 1054.895,A 0.000,B 0.000,C 90.000,E1 17.094} C_DIS
LIN {X -0.031,Y -393.853,Z 1054.892,A 0.000,B 0.000,C 90.000,E1 16.622} C_DIS
LIN {X 0.032,Y -392.656,Z 1054.890,A 0.000,B 0.000,C 90.000,E1 16.260} C_DIS
LIN {X 0.057,Y -392.208,Z 1054.889,A 0.000,B 0.000,C 90.000,E1 16.079} C_DIS
LIN {X 0.025,Y -391.551,Z 1054.886,A 0.000,B 0.000,C 90.000,E1 15.552} C_DIS
LIN {X -0.121,Y -391.637,Z 1054.883,A 0.000,B 0.000,C 90.000,E1 15.009} C_DIS
LIN {X -0.146,Y -393.020,Z 1054.875,A 0.000,B 0.000,C 90.000,E1 13.592} C_DIS
LIN {X 0.051,Y -399.717,Z 1054.850,A 0.000,B 0.000,C 90.000,E1 8.973} C_DIS
LIN {X -0.164,Y -407.418,Z 1054.829,A 0.000,B 0.000,C 90.000,E1 5.163} C_DIS
LIN {X -0.205,Y -409.716,Z 1054.823,A 0.000,B 0.000,C 90.000,E1 4.131} C_DIS
LIN {X -0.208,Y -411.759,Z 1054.819,A 0.000,B 0.000,C 90.000,E1 3.440} C_DIS
LIN {X -0.193,Y -414.208,Z 1054.816,A 0.000,B 0.000,C 90.000,E1 2.922} C_DIS
LIN {X -0.194,Y -415.143,Z 1054.815,A 0.000,B 0.000,C 90.000,E1 2.751} C_DIS
LIN {X 0.207,Y -417.266,Z 1054.814,A 0.000,B 0.000,C 90.000,E1 2.407} C_DIS
LIN {X -0.136,Y -421.668,Z 1054.811,A 0.000,B 0.000,C 90.000,E1 2.064} C_DIS
LIN {X -0.064,Y -432.646,Z 1054.807,A 0.000,B 0.000,C 90.000,E1 1.318} C_DIS
LIN {X 0.086,Y -454.812,Z 1054.799,A 0.000,B 0.000,C 90.000,E1 359.885} C_DIS
LIN {X -0.177,Y -473.027,Z 1054.793,A 0.000,B 0.000,C 90.000,E1 358.797} C_DIS
LIN {X 0.129,Y -482.860,Z 1054.790,A 0.000,B 0.000,C 90.000,E1 358.165} C_DIS
LIN {X -0.220,Y -490.945,Z 1054.787,A 0.000,B 0.000,C 90.000,E1 357.707} C_DIS
LIN {X -0.059,Y -502.050,Z 1054.783,A 0.000,B 0.000,C 90.000,E1 356.963} C_DIS
LIN {X -0.171,Y -511.276,Z 1054.780,A 0.000,B 0.000,C 90.000,E1 356.331} C_DIS
LIN {X -0.146,Y -518.815,Z 1054.776,A 0.000,B 0.000,C 90.000,E1 355.755} C_DIS
LIN {X 0.112,Y -527.489,Z 1054.772,A 0.000,B 0.000,C 90.000,E1 355.008} C_DIS
LIN {X 0.070,Y -534.429,Z 1054.769,A 0.000,B 0.000,C 90.000,E1 354.375} C_DIS
LIN {X -0.221,Y -540.872,Z 1054.765,A 0.000,B 0.000,C 90.000,E1 353.742} C_DIS
LIN {X -0.056,Y -545.876,Z 1054.762,A 0.000,B 0.000,C 90.000,E1 353.166} C_DIS
LIN {X -0.120,Y -551.500,Z 1054.758,A 0.000,B 0.000,C 90.000,E1 352.470} C_DIS
LIN {X 0.028,Y -555.672,Z 1054.755,A 0.000,B 0.000,C 90.000,E1 351.894} C_DIS
LIN {X 0.040,Y -560.262,Z 1054.751,A 0.000,B 0.000,C 90.000,E1 351.197} C_DIS
LIN {X 0.092,Y -564.458,Z 1054.747,A 0.000,B 0.000,C 90.000,E1 350.500} C_DIS
LIN {X 0.184,Y -568.229,Z 1054.744,A 0.000,B 0.000,C 90.000,E1 349.803} C_DIS
LIN {X -0.062,Y -573.095,Z 1054.738,A 0.000,B 0.000,C 90.000,E1 348.870} C_DIS
LIN {X -0.019,Y -576.833,Z 1054.734,A 0.000,B 0.000,C 90.000,E1 348.049} C_DIS
LIN {X 0.283,Y -581.498,Z 1054.728,A 0.000,B 0.000,C 90.000,E1 346.937} C_DIS
LIN {X 0.075,Y -585.780,Z 1054.722,A 0.000,B 0.000,C 90.000,E1 345.880} C_DIS
LIN {X -0.248,Y -590.911,Z 1054.714,A 0.000,B 0.000,C 90.000,E1 344.574} C_DIS
LIN {X 0.253,Y -595.809,Z 1054.707,A 0.000,B 0.000,C 90.000,E1 343.196} C_DIS
LIN {X -0.188,Y -599.419,Z 1054.701,A 0.000,B 0.000,C 90.000,E1 342.181} C_DIS
LIN {X 0.172,Y -602.807,Z 1054.695,A 0.000,B 0.000,C 90.000,E1 341.094} C_DIS
LIN {X 0.009,Y -605.895,Z 1054.689,A 0.000,B 0.000,C 90.000,E1 340.061} C_DIS
LIN {X 0.226,Y -607.351,Z 1054.686,A 0.000,B 0.000,C 90.000,E1 339.518} C_DIS
LIN {X 0.338,Y -610.157,Z 1054.681,A 0.000,B 0.000,C 90.000,E1 338.465} C_DIS
LIN {X -0.305,Y -612.712,Z 1054.675,A 0.000,B 0.000,C 90.000,E1 337.486} C_DIS
LIN {X -0.123,Y -615.077,Z 1054.669,A 0.000,B 0.000,C 90.000,E1 336.433} C_DIS
LIN {X -0.220,Y -617.177,Z 1054.663,A 0.000,B 0.000,C 90.000,E1 335.409} C_DIS
LIN {X 0.014,Y -618.977,Z 1054.658,A 0.000,B 0.000,C 90.000,E1 334.357} C_DIS
LIN {X -0.018,Y -620.219,Z 1054.653,A 0.000,B 0.000,C 90.000,E1 333.589} C_DIS
LIN {X 0.244,Y -621.995,Z 1054.646,A 0.000,B 0.000,C 90.000,E1 332.281} C_DIS
LIN {X 0.247,Y -623.330,Z 1054.641,A 0.000,B 0.000,C 90.000,E1 331.257} C_DIS
LIN {X 0.019,Y -624.448,Z 1054.635,A 0.000,B 0.000,C 90.000,E1 330.255} C_DIS
LIN {X 0.351,Y -625.297,Z 1054.629,A 0.000,B 0.000,C 90.000,E1 329.203} C_DIS
LIN {X 0.150,Y -625.822,Z 1054.625,A 0.000,B 0.000,C 90.000,E1 328.456} C_DIS
LIN {X -0.044,Y -626.456,Z 1054.618,A 0.000,B 0.000,C 90.000,E1 327.199} C_DIS
LIN {X 0.102,Y -626.598,Z 1054.612,A 0.000,B 0.000,C 90.000,E1 326.167} C_DIS
LIN {X 0.081,Y -626.570,Z 1054.605,A 0.000,B 0.000,C 90.000,E1 324.895} C_DIS
LIN {X 0.066,Y -626.343,Z 1054.598,A 0.000,B 0.000,C 90.000,E1 323.623} C_DIS
LIN {X -0.110,Y -626.019,Z 1054.589,A 0.000,B 0.000,C 90.000,E1 322.110} C_DIS
LIN {X 0.099,Y -625.790,Z 1054.581,A 0.000,B 0.000,C 90.000,E1 320.561} C_DIS
LIN {X 0.158,Y -625.661,Z 1054.571,A 0.000,B 0.000,C 90.000,E1 318.771} C_DIS
LIN {X 0.286,Y -625.446,Z 1054.563,A 0.000,B 0.000,C 90.000,E1 317.229} C_DIS
LIN {X -0.051,Y -625.248,Z 1054.554,A 0.000,B 0.000,C 90.000,E1 315.729} C_DIS
LIN {X -0.221,Y -625.045,Z 1054.543,A 0.000,B 0.000,C 90.000,E1 313.704} C_DIS
LIN {X -0.300,Y -624.913,Z 1054.537,A 0.000,B 0.000,C 90.000,E1 312.690} C_DIS
LIN {X 0.086,Y -624.639,Z 1054.531,A 0.000,B 0.000,C 90.000,E1 311.634} C_DIS
LIN {X 0.046,Y -624.200,Z 1054.521,A 0.000,B 0.000,C 90.000,E1 309.850} C_DIS
LIN {X -0.129,Y -623.817,Z 1054.514,A 0.000,B 0.000,C 90.000,E1 308.588} C_DIS
LIN {X 0.134,Y -623.652,Z 1054.506,A 0.000,B 0.000,C 90.000,E1 307.030} C_DIS
LIN {X 0.307,Y -623.533,Z 1054.503,A 0.000,B 0.000,C 90.000,E1 306.503} C_DIS
LIN {X -0.300,Y -623.469,Z 1054.495,A 0.000,B 0.000,C 90.000,E1 305.025} C_DIS
LIN {X -0.065,Y -623.696,Z 1054.484,A 0.000,B 0.000,C 90.000,E1 303.214} C_DIS
LIN {X 0.250,Y -623.722,Z 1054.482,A 0.000,B 0.000,C 90.000,E1 302.673} C_DIS
LIN {X -0.292,Y -623.942,Z 1054.479,A 0.000,B 0.000,C 90.000,E1 302.212} C_DIS
LIN {X 0.349,Y -624.193,Z 1054.473,A 0.000,B 0.000,C 90.000,E1 301.131} C_DIS
LIN {X -0.185,Y -624.187,Z 1054.470,A 0.000,B 0.000,C 90.000,E1 300.669} C_DIS
LIN {X 0.133,Y -624.449,Z 1054.469,A 0.000,B 0.000,C 90.000,E1 300.384} C_DIS
LIN {X -0.080,Y -624.982,Z 1054.462,A 0.000,B 0.000,C 90.000,E1 299.127} C_DIS
LIN {X -0.065,Y -625.049,Z 1054.459,A 0.000,B 0.000,C 90.000,E1 298.615} C_DIS
LIN {X -0.056,Y -625.276,Z 1054.458,A 0.000,B 0.000,C 90.000,E1 298.359} C_DIS
LIN {X 0.005,Y -625.523,Z 1054.450,A 0.000,B 0.000,C 90.000,E1 297.078} C_DIS
LIN {X 0.074,Y -625.341,Z 1054.443,A 0.000,B 0.000,C 90.000,E1 295.796} C_DIS
LIN {X 0.121,Y -624.910,Z 1054.438,A 0.000,B 0.000,C 90.000,E1 294.771} C_DIS
LIN {X -0.102,Y -623.951,Z 1054.432,A 0.000,B 0.000,C 90.000,E1 293.770} C_DIS
LIN {X -0.094,Y -623.065,Z 1054.428,A 0.000,B 0.000,C 90.000,E1 293.003} C_DIS
LIN {X 0.232,Y -621.878,Z 1054.424,A 0.000,B 0.000,C 90.000,E1 292.206} C_DIS
LIN {X -0.017,Y -620.708,Z 1054.421,A 0.000,B 0.000,C 90.000,E1 291.716} C_DIS
LIN {X -0.029,Y -619.996,Z 1054.419,A 0.000,B 0.000,C 90.000,E1 291.461} C_DIS
LIN {X -0.269,Y -619.120,Z 1054.418,A 0.000,B 0.000,C 90.000,E1 291.227} C_DIS
LIN {X 0.290,Y -618.036,Z 1054.416,A 0.000,B 0.000,C 90.000,E1 290.918} C_DIS
LIN {X 0.020,Y -615.097,Z 1054.414,A 0.000,B 0.000,C 90.000,E1 290.429} C_DIS
LIN {X -0.017,Y -612.920,Z 1054.412,A 0.000,B 0.000,C 90.000,E1 290.174} C_DIS
LIN {X 0.234,Y -611.369,Z 1054.411,A 0.000,B 0.000,C 90.000,E1 289.939} C_DIS
LIN {X 0.209,Y -609.946,Z 1054.410,A 0.000,B 0.000,C 90.000,E1 289.812} C_DIS
LIN {X -0.211,Y -606.355,Z 1054.409,A 0.000,B 0.000,C 90.000,E1 289.631} C_DIS
LIN {X 0.169,Y -605.447,Z 1054.408,A 0.000,B 0.000,C 90.000,E1 289.504} C_DIS
LIN {X -0.020,Y -603.835,Z 1054.408,A 0.000,B 0.000,C 90.000,E1 289.396} C_DIS
LIN {X -0.008,Y -601.630,Z 1054.407,A 0.000,B 0.000,C 90.000,E1 289.268} C_DIS
LIN {X -0.185,Y -599.686,Z 1054.407,A 0.000,B 0.000,C 90.000,E1 289.195} C_DIS
LIN {X 0.310,Y -596.874,Z 1054.406,A 0.000,B 0.000,C 90.000,E1 288.960} C_DIS
LIN {X 0.033,Y -592.122,Z 1054.404,A 0.000,B 0.000,C 90.000,E1 288.779} C_DIS
LIN {X -0.223,Y -587.982,Z 1054.403,A 0.000,B 0.000,C 90.000,E1 288.598} C_DIS
LIN {X 0.161,Y -583.751,Z 1054.402,A 0.000,B 0.000,C 90.000,E1 288.417} C_DIS
LIN {X 0.282,Y -577.867,Z 1054.401,A 0.000,B 0.000,C 90.000,E1 288.236} C_DIS
LIN {X -0.150,Y -570.769,Z 1054.401,A 0.000,B 0.000,C 90.000,E1 288.109} C_DIS
LIN {X -0.133,Y -565.406,Z 1054.400,A 0.000,B 0.000,C 90.000,E1 287.928} C_DIS
LIN {X -0.173,Y -563.081,Z 1054.399,A 0.000,B 0.000,C 90.000,E1 287.873} C_DIS
LIN {X -0.214,Y -559.888,Z 1054.399,A 0.000,B 0.000,C 90.000,E1 287.819} C_DIS
LIN {X -0.165,Y -554.695,Z 1054.399,A 0.000,B 0.000,C 90.000,E1 287.747} C_DIS
LIN {X 0.086,Y -551.064,Z 1054.398,A 0.000,B 0.000,C 90.000,E1 287.638} C_DIS
LIN {X -0.181,Y -547.447,Z 1054.397,A 0.000,B 0.000,C 90.000,E1 287.457} C_DIS
LIN {X -0.236,Y -547.417,Z 1054.397,A 0.000,B 0.000,C 90.000,E1 287.457} C_DIS
LIN {X 0.094,Y -546.829,Z 1054.396,A 0.000,B 0.000,C 90.000,E1 287.275} C_DIS
LIN {X -0.109,Y -546.160,Z 1054.393,A 0.000,B 0.000,C 90.000,E1 286.804} C_DIS
LIN {X 0.160,Y -545.025,Z 1054.378,A 0.000,B 0.000,C 90.000,E1 283.953} C_DIS
LIN {X 0.119,Y -544.553,Z 1054.371,A 0.000,B 0.000,C 90.000,E1 282.827} C_DIS
LIN {X 0.034,Y -543.788,Z 1054.364,A 0.000,B 0.000,C 90.000,E1 281.422} C_DIS
LIN {X 0.014,Y -542.748,Z 1054.354,A 0.000,B 0.000,C 90.000,E1 279.726} C_DIS
LIN {X -0.288,Y -541.918,Z 1054.346,A 0.000,B 0.000,C 90.000,E1 278.341} C_DIS
LIN {X 0.090,Y -540.539,Z 1054.334,A 0.000,B 0.000,C 90.000,E1 276.030} C_DIS
LIN {X -0.239,Y -539.508,Z 1054.324,A 0.000,B 0.000,C 90.000,E1 274.359} C_DIS
LIN {X -0.089,Y -538.398,Z 1054.313,A 0.000,B 0.000,C 90.000,E1 272.350} C_DIS
LIN {X -0.012,Y -537.581,Z 1054.305,A 0.000,B 0.000,C 90.000,E1 270.917} C_DIS
LIN {X 0.045,Y -536.542,Z 1054.296,A 0.000,B 0.000,C 90.000,E1 269.198} C_DIS
LIN {X 0.086,Y -535.649,Z 1054.288,A 0.000,B 0.000,C 90.000,E1 267.764} C_DIS
LIN {X 0.113,Y -534.674,Z 1054.280,A 0.000,B 0.000,C 90.000,E1 266.331} C_DIS
LIN {X 0.164,Y -533.895,Z 1054.273,A 0.000,B 0.000,C 90.000,E1 265.179} C_DIS
LIN {X 0.190,Y -532.824,Z 1054.265,A 0.000,B 0.000,C 90.000,E1 263.742} C_DIS
LIN {X 0.242,Y -532.079,Z 1054.261,A 0.000,B 0.000,C 90.000,E1 262.875} C_DIS
LIN {X -0.204,Y -530.208,Z 1054.251,A 0.000,B 0.000,C 90.000,E1 261.197} C_DIS
LIN {X -0.120,Y -528.733,Z 1054.243,A 0.000,B 0.000,C 90.000,E1 259.746} C_DIS
LIN {X 0.032,Y -527.116,Z 1054.235,A 0.000,B 0.000,C 90.000,E1 258.285} C_DIS
LIN {X 0.129,Y -525.875,Z 1054.229,A 0.000,B 0.000,C 90.000,E1 257.117} C_DIS
LIN {X -0.018,Y -523.727,Z 1054.217,A 0.000,B 0.000,C 90.000,E1 255.102} C_DIS
LIN {X -0.215,Y -521.926,Z 1054.208,A 0.000,B 0.000,C 90.000,E1 253.378} C_DIS
LIN {X 0.207,Y -520.352,Z 1054.199,A 0.000,B 0.000,C 90.000,E1 251.873} C_DIS
LIN {X 0.102,Y -518.676,Z 1054.191,A 0.000,B 0.000,C 90.000,E1 250.423} C_DIS
LIN {X 0.089,Y -516.542,Z 1054.182,A 0.000,B 0.000,C 90.000,E1 248.666} C_DIS
LIN {X 0.138,Y -515.067,Z 1054.175,A 0.000,B 0.000,C 90.000,E1 247.486} C_DIS
LIN {X -0.181,Y -512.964,Z 1054.167,A 0.000,B 0.000,C 90.000,E1 246.049} C_DIS
LIN {X 0.140,Y -510.742,Z 1054.159,A 0.000,B 0.000,C 90.000,E1 244.537} C_DIS
LIN {X -0.177,Y -507.850,Z 1054.149,A 0.000,B 0.000,C 90.000,E1 242.794} C_DIS
LIN {X -0.181,Y -505.330,Z 1054.141,A 0.000,B 0.000,C 90.000,E1 241.307} C_DIS
LIN {X 0.136,Y -503.220,Z 1054.134,A 0.000,B 0.000,C 90.000,E1 240.078} C_DIS
LIN {X 0.005,Y -499.355,Z 1054.122,A 0.000,B 0.000,C 90.000,E1 237.995} C_DIS
LIN {X 0.041,Y -497.100,Z 1054.116,A 0.000,B 0.000,C 90.000,E1 236.786} C_DIS
LIN {X -0.099,Y -494.702,Z 1054.109,A 0.000,B 0.000,C 90.000,E1 235.595} C_DIS
LIN {X 0.133,Y -492.314,Z 1054.102,A 0.000,B 0.000,C 90.000,E1 234.356} C_DIS
LIN {X 0.213,Y -489.554,Z 1054.095,A 0.000,B 0.000,C 90.000,E1 233.130} C_DIS
LIN {X 0.088,Y -485.986,Z 1054.087,A 0.000,B 0.000,C 90.000,E1 231.618} C_DIS
LIN {X 0.132,Y -481.118,Z 1054.075,A 0.000,B 0.000,C 90.000,E1 229.461} C_DIS
LIN {X 0.111,Y -475.908,Z 1054.061,A 0.000,B 0.000,C 90.000,E1 226.986} C_DIS
LIN {X -0.175,Y -471.589,Z 1054.049,A 0.000,B 0.000,C 90.000,E1 224.838} C_DIS
LIN {X -0.066,Y -468.444,Z 1054.040,A 0.000,B 0.000,C 90.000,E1 223.257} C_DIS
LIN {X 0.040,Y -464.648,Z 1054.030,A 0.000,B 0.000,C 90.000,E1 221.353} C_DIS
LIN {X -0.051,Y -462.690,Z 1054.025,A 0.000,B 0.000,C 90.000,E1 220.415} C_DIS
LIN {X -0.054,Y -458.694,Z 1054.014,A 0.000,B 0.000,C 90.000,E1 218.508} C_DIS
LIN {X 0.082,Y -454.096,Z 1054.001,A 0.000,B 0.000,C 90.000,E1 216.251} C_DIS
LIN {X -0.058,Y -450.762,Z 1053.993,A 0.000,B 0.000,C 90.000,E1 214.659} C_DIS
LIN {X -0.266,Y -446.074,Z 1053.980,A 0.000,B 0.000,C 90.000,E1 212.418} C_DIS
LIN {X -0.003,Y -443.292,Z 1053.973,A 0.000,B 0.000,C 90.000,E1 211.082} C_DIS
LIN {X -0.123,Y -439.772,Z 1053.964,A 0.000,B 0.000,C 90.000,E1 209.461} C_DIS
LIN {X -0.091,Y -433.494,Z 1053.947,A 0.000,B 0.000,C 90.000,E1 206.488} C_DIS
LIN {X -0.065,Y -430.043,Z 1053.938,A 0.000,B 0.000,C 90.000,E1 204.823} C_DIS
LIN {X -0.114,Y -424.973,Z 1053.923,A 0.000,B 0.000,C 90.000,E1 202.153} C_DIS
LIN {X 0.212,Y -418.970,Z 1053.901,A 0.000,B 0.000,C 90.000,E1 198.055} C_DIS
LIN {X -0.016,Y -417.581,Z 1053.891,A 0.000,B 0.000,C 90.000,E1 196.386} C_DIS
LIN {X -0.059,Y -417.127,Z 1053.885,A 0.000,B 0.000,C 90.000,E1 195.371} C_DIS
LIN {X 0.140,Y -417.275,Z 1053.882,A 0.000,B 0.000,C 90.000,E1 194.662} C_DIS
LIN {X 0.088,Y -418.163,Z 1053.876,A 0.000,B 0.000,C 90.000,E1 193.647} C_DIS
LIN {X -0.211,Y -419.398,Z 1053.872,A 0.000,B 0.000,C 90.000,E1 193.008} C_DIS
LIN {X 0.138,Y -421.834,Z 1053.867,A 0.000,B 0.000,C 90.000,E1 192.119} C_DIS
LIN {X 0.069,Y -424.589,Z 1053.864,A 0.000,B 0.000,C 90.000,E1 191.478} C_DIS
LIN {X -0.177,Y -428.044,Z 1053.860,A 0.000,B 0.000,C 90.000,E1 190.838} C_DIS
LIN {X 0.145,Y -433.889,Z 1053.855,A 0.000,B 0.000,C 90.000,E1 189.792} C_DIS
LIN {X -0.176,Y -448.908,Z 1053.842,A 0.000,B 0.000,C 90.000,E1 187.530} C_DIS
LIN {X 0.118,Y -457.711,Z 1053.835,A 0.000,B 0.000,C 90.000,E1 186.201} C_DIS
LIN {X -0.159,Y -464.130,Z 1053.829,A 0.000,B 0.000,C 90.000,E1 185.277} C_DIS
LIN {X 0.057,Y -470.264,Z 1053.824,A 0.000,B 0.000,C 90.000,E1 184.302} C_DIS
LIN {X 0.008,Y -477.144,Z 1053.818,A 0.000,B 0.000,C 90.000,E1 183.212} C_DIS
LIN {X -0.128,Y -485.752,Z 1053.810,A 0.000,B 0.000,C 90.000,E1 181.835} C_DIS
END
